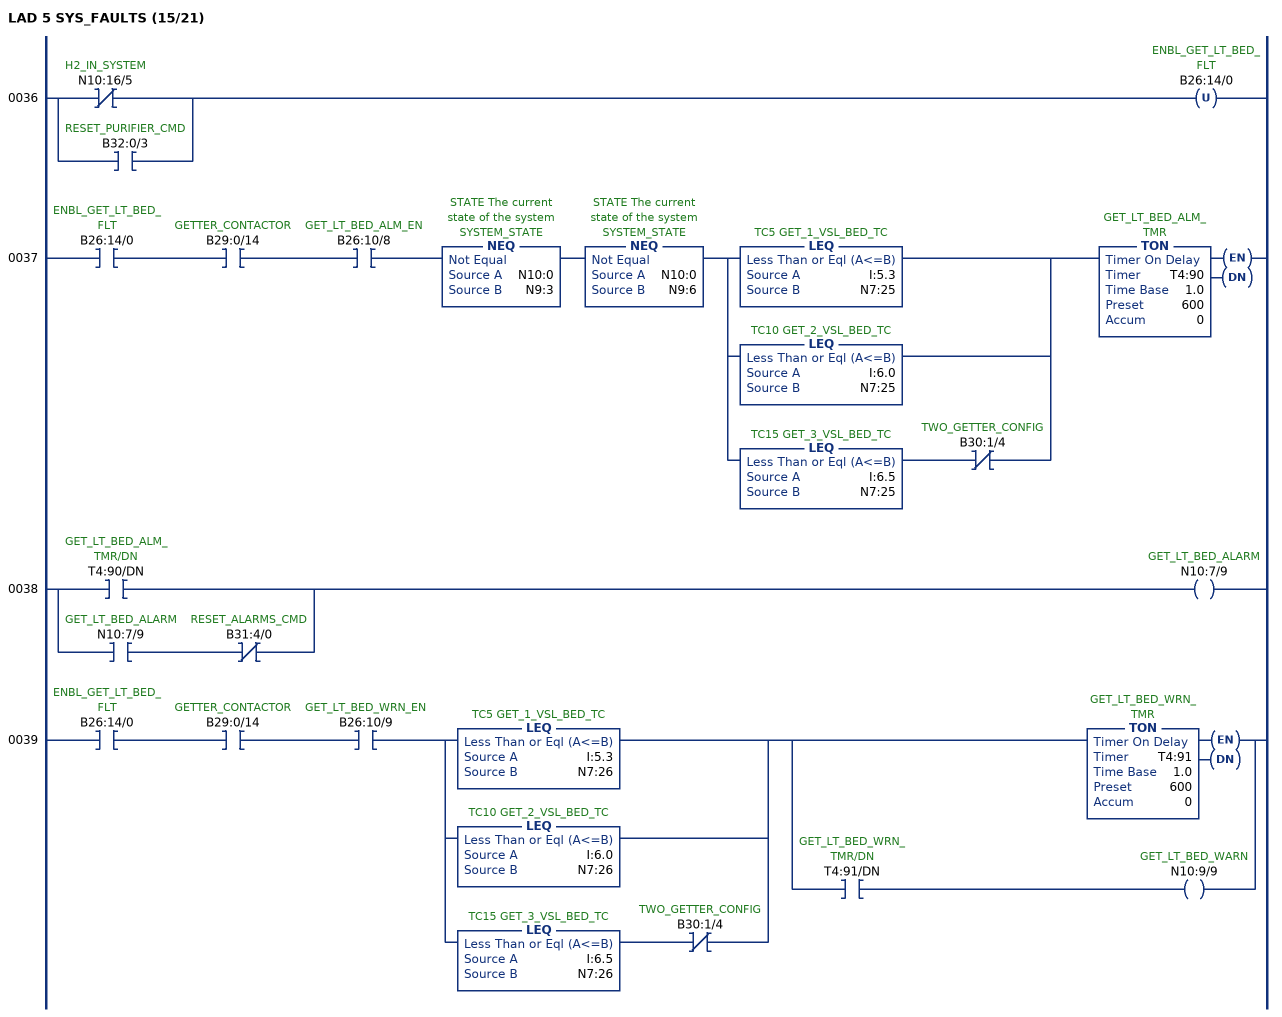
% Rung: 36 %
SOR BST XIO N10:16/5 NXB XIC B32:0/3 BND OTU B26:14/0 EOR
%   N10:16/5  H2_IN_SYSTEM %
%   B32:0/3  RESET_PURIFIER_CMD %
%   B26:14/0  ENBL_GET_LT_BED_FLT %
% Rung: 37 %
SOR XIC B26:14/0 XIC B29:0/14 XIC B26:10/8 NEQ N10:0 N9:3 NEQ N10:0 N9:6 BST LEQ I:5.3 N7:25 NXB LEQ I:6.0 N7:25 NXB LEQ I:6.5 N7:25 XIO B30:1/4 BND TON T4:90 1.0 600 0 EOR
%   B26:14/0  ENBL_GET_LT_BED_FLT %
%   B29:0/14  GETTER_CONTACTOR %
%   B26:10/8  GET_LT_BED_ALM_EN %
%   N10:0  SYSTEM_STATE  "STATE The current state of the system" %
%   N9:3  SYSTEM_MANUAL  "STATE System Manual" %
%   N9:6  SYSTEM_PURGE %
%   I:5.3  GET_1_VSL_BED_TC  "TC5" %
%   N7:25  GET_LT_BED_ALM_SP %
%   I:6.0  GET_2_VSL_BED_TC  "TC10" %
%   I:6.5  GET_3_VSL_BED_TC  "TC15" %
%   B30:1/4  TWO_GETTER_CONFIG %
%   T4:90  GET_LT_BED_ALM_TMR %
% Rung: 38 %
SOR BST XIC T4:90/DN NXB XIC N10:7/9 XIO B31:4/0 BND OTE N10:7/9 EOR
%   T4:90  GET_LT_BED_ALM_TMR %
%   N10:7/9  GET_LT_BED_ALARM %
%   B31:4/0  RESET_ALARMS_CMD %
% Rung: 39 %
SOR XIC B26:14/0 XIC B29:0/14 XIC B26:10/9 BST LEQ I:5.3 N7:26 NXB LEQ I:6.0 N7:26 NXB LEQ I:6.5 N7:26 XIO B30:1/4 BND BST TON T4:91 1.0 600 0 NXB XIC T4:91/DN OTE N10:9/9 BND EOR
%   B26:14/0  ENBL_GET_LT_BED_FLT %
%   B29:0/14  GETTER_CONTACTOR %
%   B26:10/9  GET_LT_BED_WRN_EN %
%   I:5.3  GET_1_VSL_BED_TC  "TC5" %
%   N7:26  GET_LT_BED_WRN_SP %
%   I:6.0  GET_2_VSL_BED_TC  "TC10" %
%   I:6.5  GET_3_VSL_BED_TC  "TC15" %
%   B30:1/4  TWO_GETTER_CONFIG %
%   T4:91  GET_LT_BED_WRN_TMR %
%   N10:9/9  GET_LT_BED_WARN %

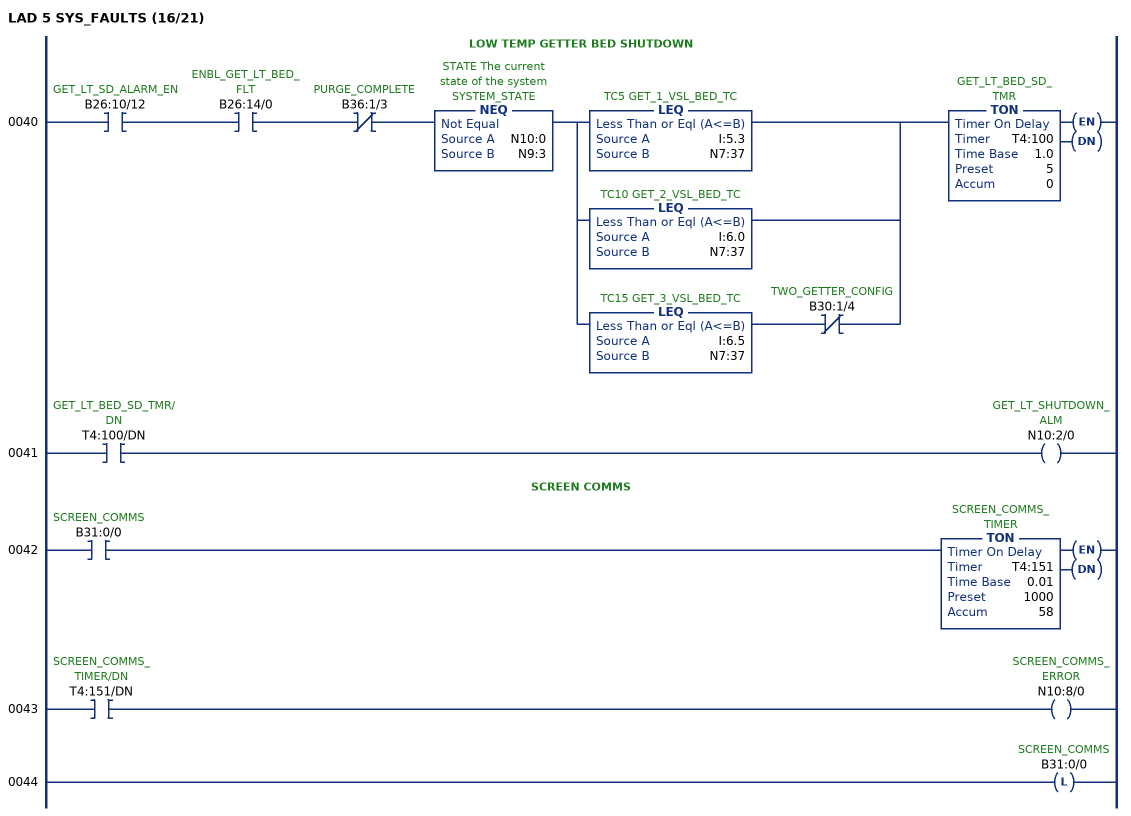
% Rung: 40 %
% TITLE: LOW TEMP GETTER BED SHUTDOWN %
SOR XIC B26:10/12 XIC B26:14/0 XIO B36:1/3 NEQ N10:0 N9:3 BST LEQ I:5.3 N7:37 NXB LEQ I:6.0 N7:37 NXB LEQ I:6.5 N7:37 XIO B30:1/4 BND TON T4:100 1.0 5 0 EOR
%   B26:10/12  GET_LT_SD_ALARM_EN %
%   B26:14/0  ENBL_GET_LT_BED_FLT %
%   B36:1/3  PURGE_COMPLETE %
%   N10:0  SYSTEM_STATE  "STATE The current state of the system" %
%   N9:3  SYSTEM_MANUAL  "STATE System Manual" %
%   I:5.3  GET_1_VSL_BED_TC  "TC5" %
%   N7:37  GET_LT_SHUTDOWN_SP %
%   I:6.0  GET_2_VSL_BED_TC  "TC10" %
%   I:6.5  GET_3_VSL_BED_TC  "TC15" %
%   B30:1/4  TWO_GETTER_CONFIG %
%   T4:100  GET_LT_BED_SD_TMR %
% Rung: 41 %
SOR XIC T4:100/DN OTE N10:2/0 EOR
%   T4:100  GET_LT_BED_SD_TMR %
%   N10:2/0  GET_LT_SHUTDOWN_ALM %
% Rung: 42 %
% TITLE: SCREEN COMMS %
SOR XIC B31:0/0 TON T4:151 0.01 1000 58 EOR
%   B31:0/0  SCREEN_COMMS %
%   T4:151  SCREEN_COMMS_TIMER %
% Rung: 43 %
SOR XIC T4:151/DN OTE N10:8/0 EOR
%   T4:151  SCREEN_COMMS_TIMER %
%   N10:8/0  SCREEN_COMMS_ERROR %
% Rung: 44 %
SOR OTL B31:0/0 EOR
%   B31:0/0  SCREEN_COMMS %

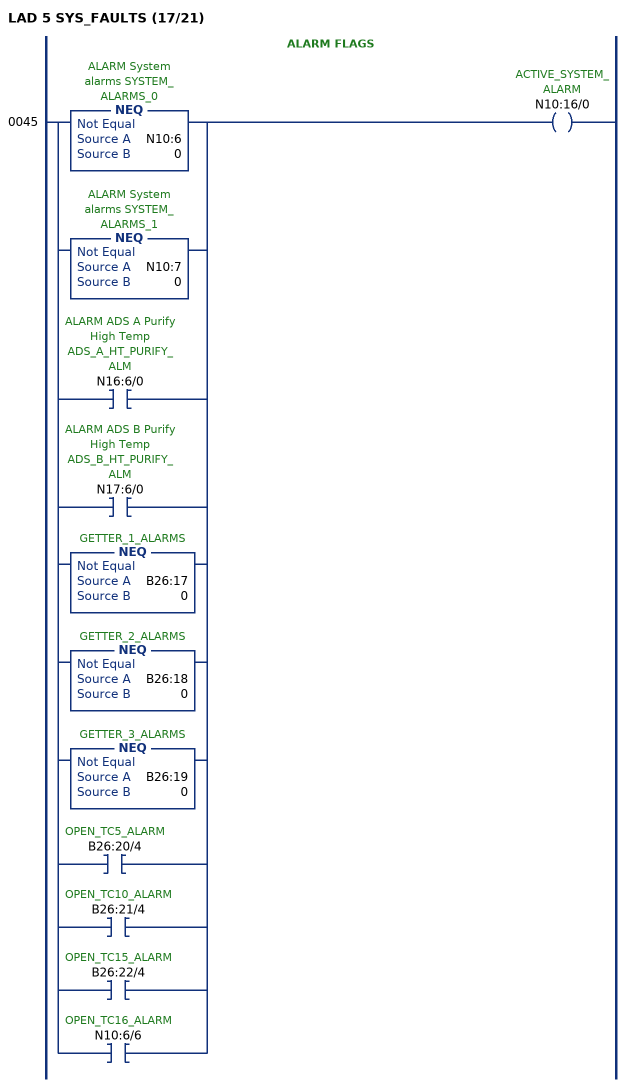
% Rung: 45 %
% TITLE: ALARM FLAGS %
SOR BST NEQ N10:6 0 NXB NEQ N10:7 0 NXB XIC N16:6/0 NXB XIC N17:6/0 NXB NEQ B26:17 0 NXB NEQ B26:18 0 NXB NEQ B26:19 0 NXB XIC B26:20/4 NXB XIC B26:21/4 NXB XIC B26:22/4 NXB XIC N10:6/6 BND OTE N10:16/0 EOR
%   N10:6  SYSTEM_ALARMS_0  "ALARM System alarms" %
%   N10:7  SYSTEM_ALARMS_1  "ALARM System alarms" %
%   N16:6/0  ADS_A_HT_PURIFY_ALM  "ALARM ADS A Purify High Temp" %
%   N17:6/0  ADS_B_HT_PURIFY_ALM  "ALARM ADS B Purify High Temp" %
%   B26:17  GETTER_1_ALARMS %
%   B26:18  GETTER_2_ALARMS %
%   B26:19  GETTER_3_ALARMS %
%   B26:20/4  OPEN_TC5_ALARM %
%   B26:21/4  OPEN_TC10_ALARM %
%   B26:22/4  OPEN_TC15_ALARM %
%   N10:6/6  OPEN_TC16_ALARM %
%   N10:16/0  ACTIVE_SYSTEM_ALARM %

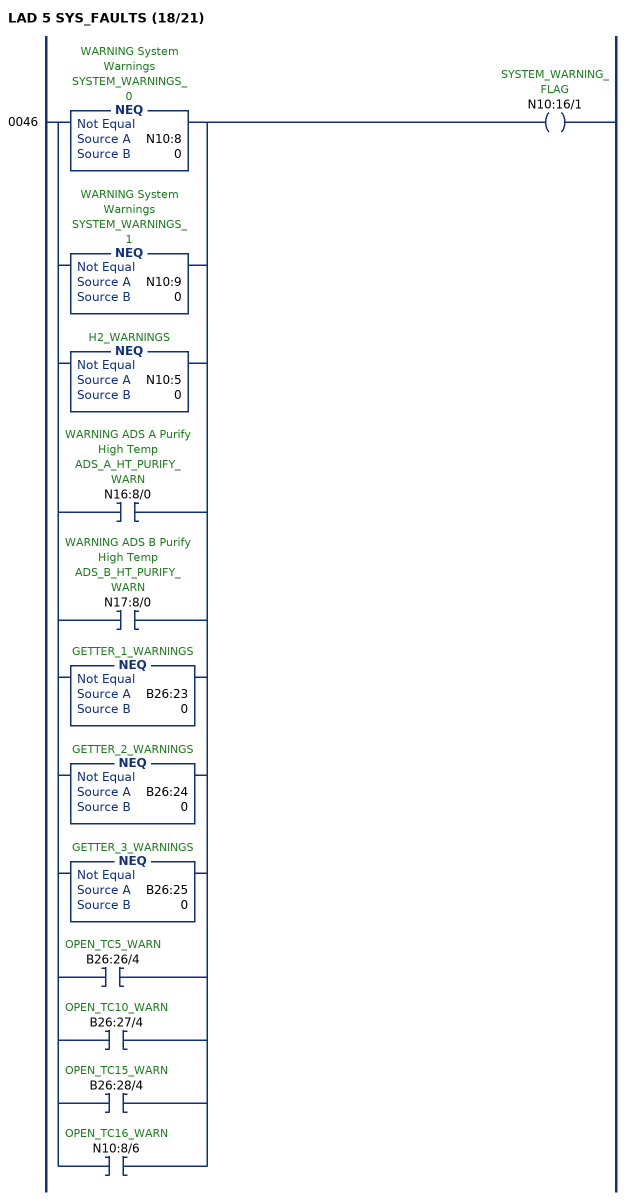
% Rung: 46 %
SOR BST NEQ N10:8 0 NXB NEQ N10:9 0 NXB NEQ N10:5 0 NXB XIC N16:8/0 NXB XIC N17:8/0 NXB NEQ B26:23 0 NXB NEQ B26:24 0 NXB NEQ B26:25 0 NXB XIC B26:26/4 NXB XIC B26:27/4 NXB XIC B26:28/4 NXB XIC N10:8/6 BND OTE N10:16/1 EOR
%   N10:8  SYSTEM_WARNINGS_0  "WARNING System Warnings" %
%   N10:9  SYSTEM_WARNINGS_1  "WARNING System Warnings" %
%   N10:5  H2_WARNINGS %
%   N16:8/0  ADS_A_HT_PURIFY_WARN  "WARNING ADS A Purify High Temp" %
%   N17:8/0  ADS_B_HT_PURIFY_WARN  "WARNING ADS B Purify High Temp" %
%   B26:23  GETTER_1_WARNINGS %
%   B26:24  GETTER_2_WARNINGS %
%   B26:25  GETTER_3_WARNINGS %
%   B26:26/4  OPEN_TC5_WARN %
%   B26:27/4  OPEN_TC10_WARN %
%   B26:28/4  OPEN_TC15_WARN %
%   N10:8/6  OPEN_TC16_WARN %
%   N10:16/1  SYSTEM_WARNING_FLAG %

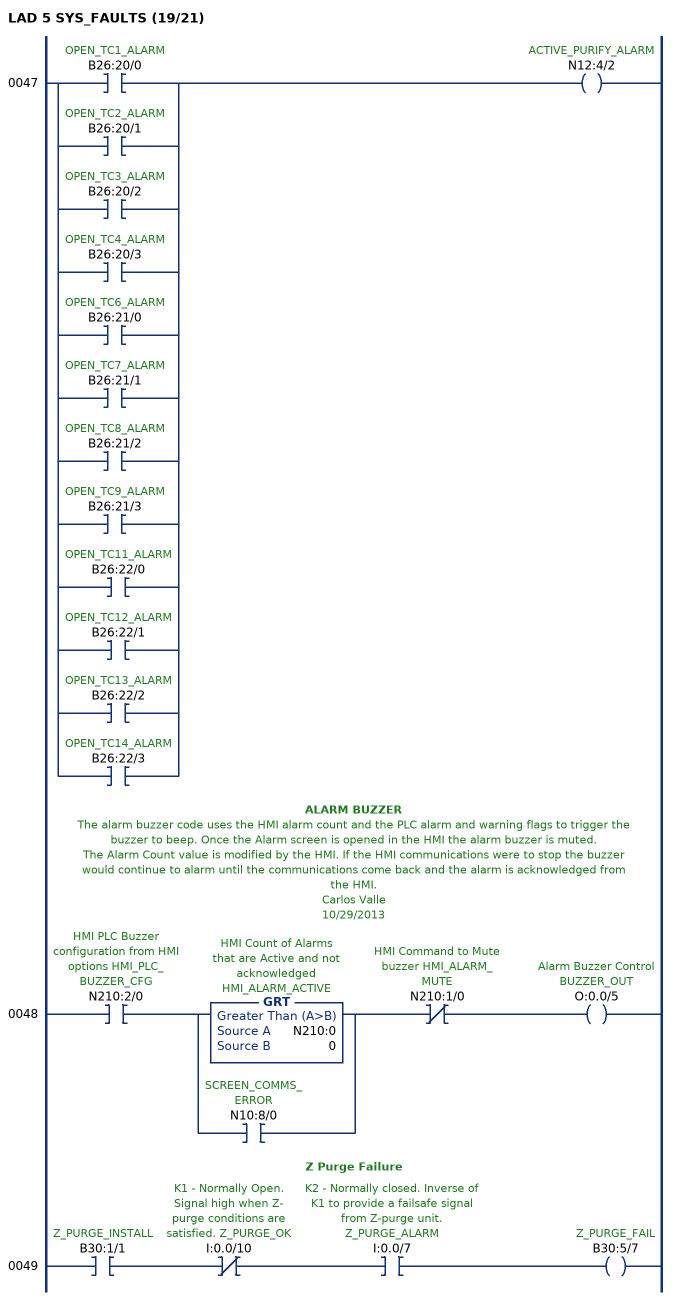
% Rung: 47 %
SOR BST XIC B26:20/0 NXB XIC B26:20/1 NXB XIC B26:20/2 NXB XIC B26:20/3 NXB XIC B26:21/0 NXB XIC B26:21/1 NXB XIC B26:21/2 NXB XIC B26:21/3 NXB XIC B26:22/0 NXB XIC B26:22/1 NXB XIC B26:22/2 NXB XIC B26:22/3 BND OTE N12:4/2 EOR
%   B26:20/0  OPEN_TC1_ALARM %
%   B26:20/1  OPEN_TC2_ALARM %
%   B26:20/2  OPEN_TC3_ALARM %
%   B26:20/3  OPEN_TC4_ALARM %
%   B26:21/0  OPEN_TC6_ALARM %
%   B26:21/1  OPEN_TC7_ALARM %
%   B26:21/2  OPEN_TC8_ALARM %
%   B26:21/3  OPEN_TC9_ALARM %
%   B26:22/0  OPEN_TC11_ALARM %
%   B26:22/1  OPEN_TC12_ALARM %
%   B26:22/2  OPEN_TC13_ALARM %
%   B26:22/3  OPEN_TC14_ALARM %
%   N12:4/2  ACTIVE_PURIFY_ALARM %
% Rung: 48 %
% TITLE: ALARM BUZZER %
% The alarm buzzer code uses the HMI alarm count and the PLC alarm and warning flags to trigger the buzzer to beep. Once the Alarm screen is opened in the HMI the alarm buzzer is muted.
% The Alarm Count value is modified by the HMI. If the HMI communications were to stop the buzzer would continue to alarm until the communications come back and the alarm is acknowledged from the HMI.
% Carlos Valle
% 10/29/2013 %
SOR XIC N210:2/0 BST GRT N210:0 0 NXB XIC N10:8/0 BND XIO N210:1/0 OTE O:0.0/5 EOR
%   N210:2/0  HMI_PLC_BUZZER_CFG  "HMI PLC Buzzer configuration from HMI options" %
%   N210:0  HMI_ALARM_ACTIVE  "HMI Count of Alarms that are Active and not acknowledged" %
%   N10:8/0  SCREEN_COMMS_ERROR %
%   N210:1/0  HMI_ALARM_MUTE  "HMI Command to Mute buzzer" %
%   O:0.0/5  BUZZER_OUT  "Alarm Buzzer Control" %
% Rung: 49 %
% TITLE: Z Purge Failure %
SOR XIC B30:1/1 XIO I:0.0/10 XIC I:0.0/7 OTE B30:5/7 EOR
%   B30:1/1  Z_PURGE_INSTALL %
%   I:0.0/10  Z_PURGE_OK  "K1 - Normally Open. Signal high when Z- purge conditions are satisfied." %
%   I:0.0/7  Z_PURGE_ALARM  "K2 - Normally closed. Inverse of K1 to provide a failsafe signal from Z-purge unit." %
%   B30:5/7  Z_PURGE_FAIL %

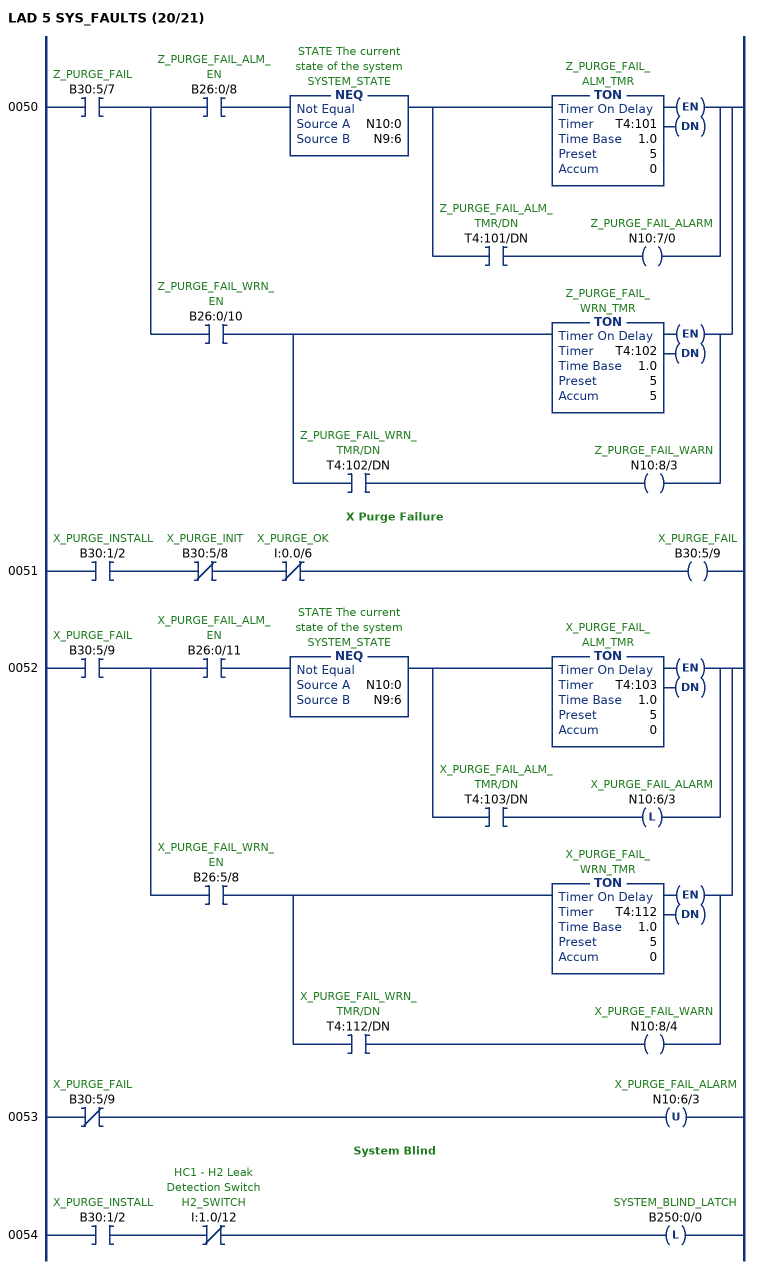
% Rung: 50 %
SOR XIC B30:5/7 BST XIC B26:0/8 NEQ N10:0 N9:6 BST TON T4:101 1.0 5 0 NXB XIC T4:101/DN OTE N10:7/0 BND NXB XIC B26:0/10 BST TON T4:102 1.0 5 5 NXB XIC T4:102/DN OTE N10:8/3 BND BND EOR
%   B30:5/7  Z_PURGE_FAIL %
%   B26:0/8  Z_PURGE_FAIL_ALM_EN %
%   N10:0  SYSTEM_STATE  "STATE The current state of the system" %
%   N9:6  SYSTEM_PURGE %
%   T4:101  Z_PURGE_FAIL_ALM_TMR %
%   N10:7/0  Z_PURGE_FAIL_ALARM %
%   B26:0/10  Z_PURGE_FAIL_WRN_EN %
%   T4:102  Z_PURGE_FAIL_WRN_TMR %
%   N10:8/3  Z_PURGE_FAIL_WARN %
% Rung: 51 %
% TITLE: X Purge Failure %
SOR XIC B30:1/2 XIO B30:5/8 XIO I:0.0/6 OTE B30:5/9 EOR
%   B30:1/2  X_PURGE_INSTALL %
%   B30:5/8  X_PURGE_INIT %
%   I:0.0/6  X_PURGE_OK %
%   B30:5/9  X_PURGE_FAIL %
% Rung: 52 %
SOR XIC B30:5/9 BST XIC B26:0/11 NEQ N10:0 N9:6 BST TON T4:103 1.0 5 0 NXB XIC T4:103/DN OTL N10:6/3 BND NXB XIC B26:5/8 BST TON T4:112 1.0 5 0 NXB XIC T4:112/DN OTE N10:8/4 BND BND EOR
%   B30:5/9  X_PURGE_FAIL %
%   B26:0/11  X_PURGE_FAIL_ALM_EN %
%   N10:0  SYSTEM_STATE  "STATE The current state of the system" %
%   N9:6  SYSTEM_PURGE %
%   T4:103  X_PURGE_FAIL_ALM_TMR %
%   N10:6/3  X_PURGE_FAIL_ALARM %
%   B26:5/8  X_PURGE_FAIL_WRN_EN %
%   T4:112  X_PURGE_FAIL_WRN_TMR %
%   N10:8/4  X_PURGE_FAIL_WARN %
% Rung: 53 %
SOR XIO B30:5/9 OTU N10:6/3 EOR
%   B30:5/9  X_PURGE_FAIL %
%   N10:6/3  X_PURGE_FAIL_ALARM %
% Rung: 54 %
% TITLE: System Blind %
SOR XIC B30:1/2 XIO I:1.0/12 OTL B250:0/0 EOR
%   B30:1/2  X_PURGE_INSTALL %
%   I:1.0/12  H2_SWITCH  "HC1 - H2 Leak Detection Switch" %
%   B250:0/0  SYSTEM_BLIND_LATCH %

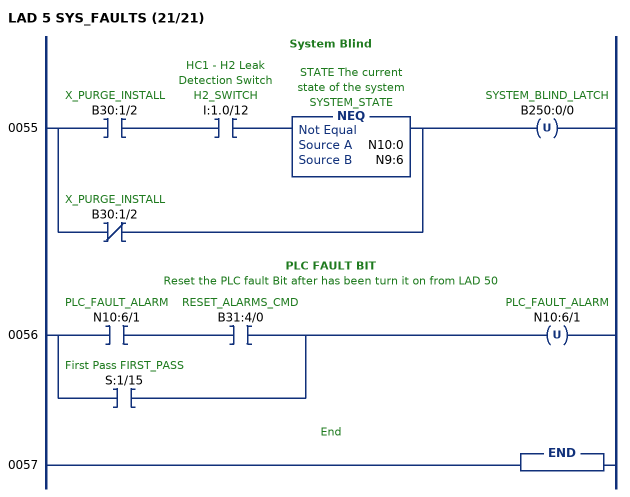
% Rung: 55 %
% TITLE: System Blind %
SOR BST XIC B30:1/2 XIC I:1.0/12 NEQ N10:0 N9:6 NXB XIO B30:1/2 BND OTU B250:0/0 EOR
%   B30:1/2  X_PURGE_INSTALL %
%   I:1.0/12  H2_SWITCH  "HC1 - H2 Leak Detection Switch" %
%   N10:0  SYSTEM_STATE  "STATE The current state of the system" %
%   N9:6  SYSTEM_PURGE %
%   B250:0/0  SYSTEM_BLIND_LATCH %
% Rung: 56 %
% TITLE: PLC FAULT BIT %
% Reset the PLC fault Bit after has been turn it on from LAD 50 %
SOR BST XIC N10:6/1 XIC B31:4/0 NXB XIC S:1/15 BND OTU N10:6/1 EOR
%   N10:6/1  PLC_FAULT_ALARM %
%   B31:4/0  RESET_ALARMS_CMD %
%   S:1/15  FIRST_PASS  "First Pass" %
% Rung: 57 %
% End %
SOR END EOR

LADDER 6 "SYSTEM"    % Controls the system %
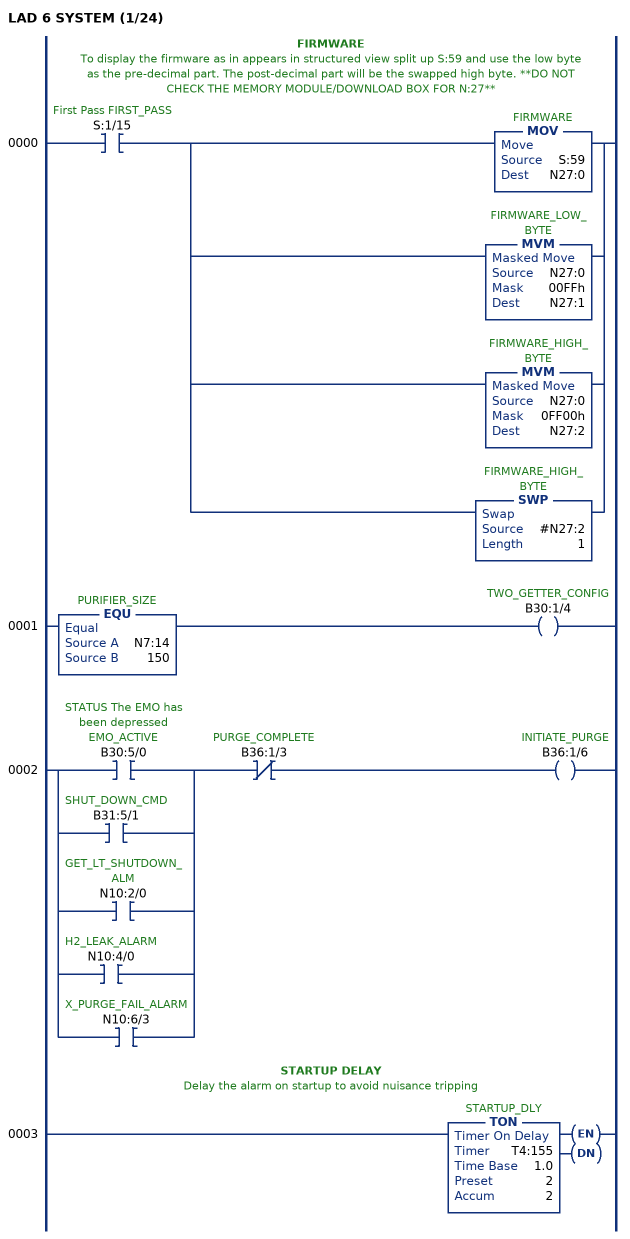
% Rung: 0 %
% TITLE: FIRMWARE %
% To display the firmware as in appears in structured view split up S:59 and use the low byte as the pre-decimal part. The post-decimal part will be the swapped high byte. **DO NOT CHECK THE MEMORY MODULE/DOWNLOAD BOX FOR N:27** %
SOR XIC S:1/15 BST MOV S:59 N27:0 NXB MVM N27:0 00FFh N27:1 NXB MVM N27:0 0FF00h N27:2 NXB SWP #N27:2 1 BND EOR
%   S:1/15  FIRST_PASS  "First Pass" %
%   S:59  "Operating System FRN" %
%   N27:0  FIRMWARE %
%   N27:1  FIRMWARE_LOW_BYTE %
%   N27:2  FIRMWARE_HIGH_BYTE %
% Rung: 1 %
SOR EQU N7:14 150 OTE B30:1/4 EOR
%   N7:14  PURIFIER_SIZE %
%   B30:1/4  TWO_GETTER_CONFIG %
% Rung: 2 %
SOR BST XIC B30:5/0 NXB XIC B31:5/1 NXB XIC N10:2/0 NXB XIC N10:4/0 NXB XIC N10:6/3 BND XIO B36:1/3 OTE B36:1/6 EOR
%   B30:5/0  EMO_ACTIVE  "STATUS The EMO has been depressed" %
%   B31:5/1  SHUT_DOWN_CMD %
%   N10:2/0  GET_LT_SHUTDOWN_ALM %
%   N10:4/0  H2_LEAK_ALARM %
%   N10:6/3  X_PURGE_FAIL_ALARM %
%   B36:1/3  PURGE_COMPLETE %
%   B36:1/6  INITIATE_PURGE %
% Rung: 3 %
% TITLE: STARTUP DELAY %
% Delay the alarm on startup to avoid nuisance tripping %
SOR TON T4:155 1.0 2 2 EOR
%   T4:155  STARTUP_DLY %

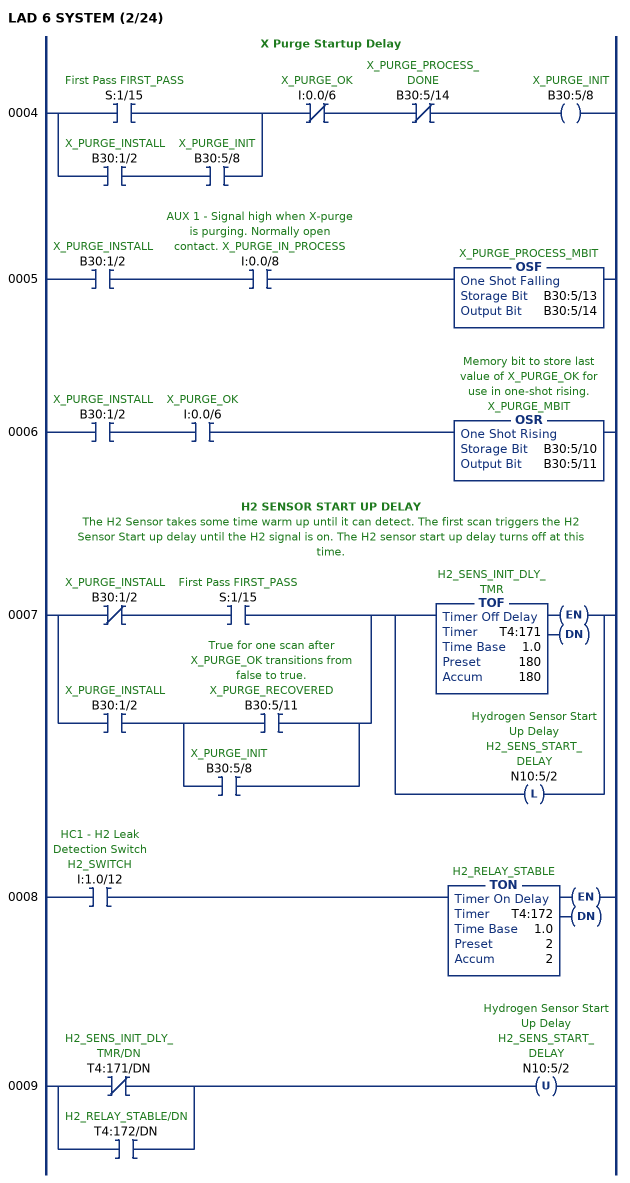
% Rung: 4 %
% TITLE: X Purge Startup Delay %
SOR BST XIC S:1/15 NXB XIC B30:1/2 XIC B30:5/8 BND XIO I:0.0/6 XIO B30:5/14 OTE B30:5/8 EOR
%   S:1/15  FIRST_PASS  "First Pass" %
%   B30:1/2  X_PURGE_INSTALL %
%   B30:5/8  X_PURGE_INIT %
%   I:0.0/6  X_PURGE_OK %
%   B30:5/14  X_PURGE_PROCESS_DONE %
% Rung: 5 %
SOR XIC B30:1/2 XIC I:0.0/8 OSF B30:5/13 B30:5/14 EOR
%   B30:1/2  X_PURGE_INSTALL %
%   I:0.0/8  X_PURGE_IN_PROCESS  "AUX 1 - Signal high when X-purge is purging. Normally open contact." %
%   B30:5/13  X_PURGE_PROCESS_MBIT %
%   B30:5/14  X_PURGE_PROCESS_DONE %
% Rung: 6 %
SOR XIC B30:1/2 XIC I:0.0/6 OSR B30:5/10 B30:5/11 EOR
%   B30:1/2  X_PURGE_INSTALL %
%   I:0.0/6  X_PURGE_OK %
%   B30:5/10  X_PURGE_MBIT  "Memory bit to store last value of X_PURGE_OK for use in one-shot rising." %
%   B30:5/11  X_PURGE_RECOVERED  "True for one scan after X_PURGE_OK transitions from false to true." %
% Rung: 7 %
% TITLE: H2 SENSOR START UP DELAY %
% The H2 Sensor takes some time warm up until it can detect. The first scan triggers the H2 Sensor Start up delay until the H2 signal is on. The H2 sensor start up delay turns off at this time. %
SOR BST XIO B30:1/2 XIC S:1/15 NXB XIC B30:1/2 BST XIC B30:5/11 NXB XIC B30:5/8 BND BND BST TOF T4:171 1.0 180 180 NXB OTL N10:5/2 BND EOR
%   B30:1/2  X_PURGE_INSTALL %
%   S:1/15  FIRST_PASS  "First Pass" %
%   B30:5/11  X_PURGE_RECOVERED  "True for one scan after X_PURGE_OK transitions from false to true." %
%   B30:5/8  X_PURGE_INIT %
%   T4:171  H2_SENS_INIT_DLY_TMR %
%   N10:5/2  H2_SENS_START_DELAY  "Hydrogen Sensor Start Up Delay" %
% Rung: 8 %
SOR XIC I:1.0/12 TON T4:172 1.0 2 2 EOR
%   I:1.0/12  H2_SWITCH  "HC1 - H2 Leak Detection Switch" %
%   T4:172  H2_RELAY_STABLE %
% Rung: 9 %
SOR BST XIO T4:171/DN NXB XIC T4:172/DN BND OTU N10:5/2 EOR
%   T4:171  H2_SENS_INIT_DLY_TMR %
%   T4:172  H2_RELAY_STABLE %
%   N10:5/2  H2_SENS_START_DELAY  "Hydrogen Sensor Start Up Delay" %

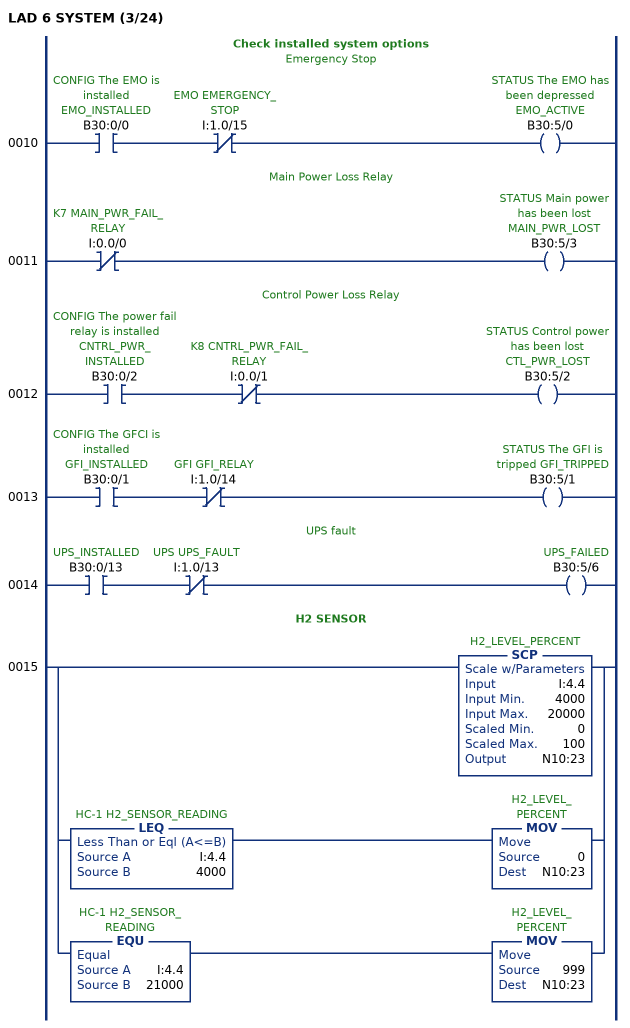
% Rung: 10 %
% TITLE: Check installed system options %
% Emergency Stop %
SOR XIC B30:0/0 XIO I:1.0/15 OTE B30:5/0 EOR
%   B30:0/0  EMO_INSTALLED  "CONFIG The EMO is installed" %
%   I:1.0/15  EMERGENCY_STOP  "EMO" %
%   B30:5/0  EMO_ACTIVE  "STATUS The EMO has been depressed" %
% Rung: 11 %
% Main Power Loss Relay %
SOR XIO I:0.0/0 OTE B30:5/3 EOR
%   I:0.0/0  MAIN_PWR_FAIL_RELAY  "K7" %
%   B30:5/3  MAIN_PWR_LOST  "STATUS Main power has been lost" %
% Rung: 12 %
% Control Power Loss Relay %
SOR XIC B30:0/2 XIO I:0.0/1 OTE B30:5/2 EOR
%   B30:0/2  CNTRL_PWR_INSTALLED  "CONFIG The power fail relay is installed" %
%   I:0.0/1  CNTRL_PWR_FAIL_RELAY  "K8" %
%   B30:5/2  CTL_PWR_LOST  "STATUS Control power has been lost" %
% Rung: 13 %
SOR XIC B30:0/1 XIO I:1.0/14 OTE B30:5/1 EOR
%   B30:0/1  GFI_INSTALLED  "CONFIG The GFCI is installed" %
%   I:1.0/14  GFI_RELAY  "GFI" %
%   B30:5/1  GFI_TRIPPED  "STATUS The GFI is tripped" %
% Rung: 14 %
% UPS fault %
SOR XIC B30:0/13 XIO I:1.0/13 OTE B30:5/6 EOR
%   B30:0/13  UPS_INSTALLED %
%   I:1.0/13  UPS_FAULT  "UPS" %
%   B30:5/6  UPS_FAILED %
% Rung: 15 %
% TITLE: H2 SENSOR %
SOR BST SCP I:4.4 4000 20000 0 100 N10:23 NXB LEQ I:4.4 4000 MOV 0 N10:23 NXB EQU I:4.4 21000 MOV 999 N10:23 BND EOR
%   I:4.4  H2_SENSOR_READING  "HC-1" %
%   N10:23  H2_LEVEL_PERCENT %

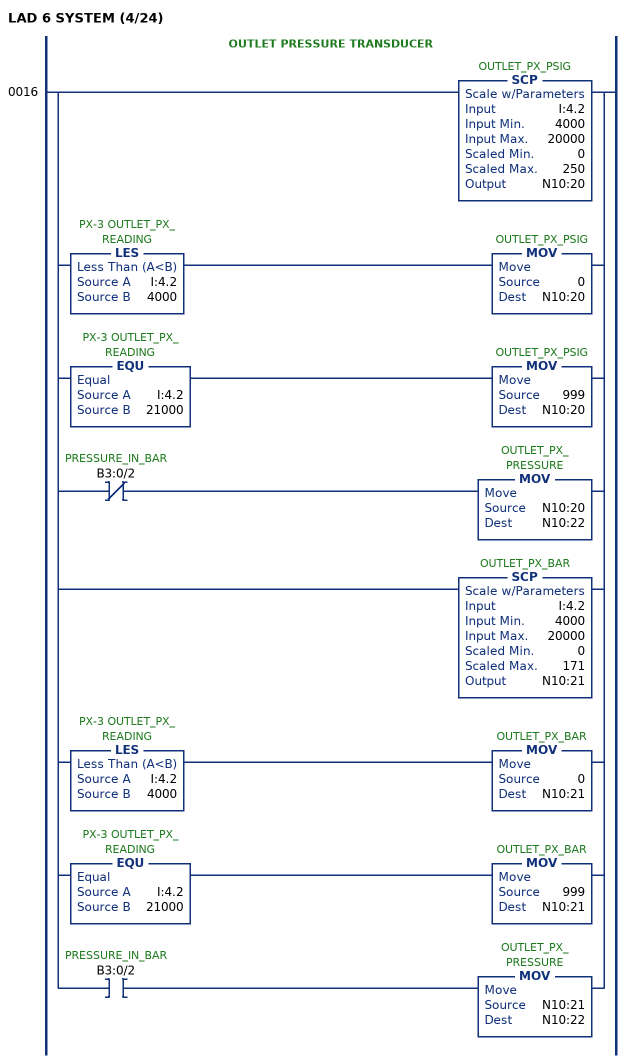
% Rung: 16 %
% TITLE: OUTLET PRESSURE TRANSDUCER %
SOR BST SCP I:4.2 4000 20000 0 250 N10:20 NXB LES I:4.2 4000 MOV 0 N10:20 NXB EQU I:4.2 21000 MOV 999 N10:20 NXB XIO B3:0/2 MOV N10:20 N10:22 NXB SCP I:4.2 4000 20000 0 171 N10:21 NXB LES I:4.2 4000 MOV 0 N10:21 NXB EQU I:4.2 21000 MOV 999 N10:21 NXB XIC B3:0/2 MOV N10:21 N10:22 BND EOR
%   I:4.2  OUTLET_PX_READING  "PX-3" %
%   N10:20  OUTLET_PX_PSIG %
%   B3:0/2  PRESSURE_IN_BAR %
%   N10:22  OUTLET_PX_PRESSURE %
%   N10:21  OUTLET_PX_BAR %

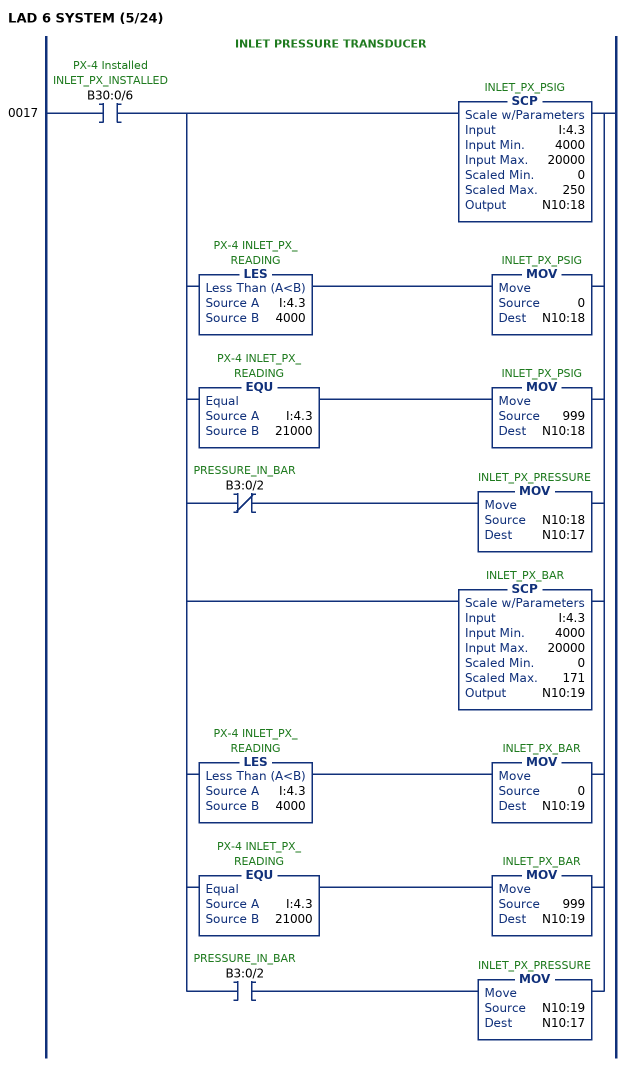
% Rung: 17 %
% TITLE: INLET PRESSURE TRANSDUCER %
SOR XIC B30:0/6 BST SCP I:4.3 4000 20000 0 250 N10:18 NXB LES I:4.3 4000 MOV 0 N10:18 NXB EQU I:4.3 21000 MOV 999 N10:18 NXB XIO B3:0/2 MOV N10:18 N10:17 NXB SCP I:4.3 4000 20000 0 171 N10:19 NXB LES I:4.3 4000 MOV 0 N10:19 NXB EQU I:4.3 21000 MOV 999 N10:19 NXB XIC B3:0/2 MOV N10:19 N10:17 BND EOR
%   B30:0/6  INLET_PX_INSTALLED  "PX-4 Installed" %
%   I:4.3  INLET_PX_READING  "PX-4" %
%   N10:18  INLET_PX_PSIG %
%   B3:0/2  PRESSURE_IN_BAR %
%   N10:17  INLET_PX_PRESSURE %
%   N10:19  INLET_PX_BAR %

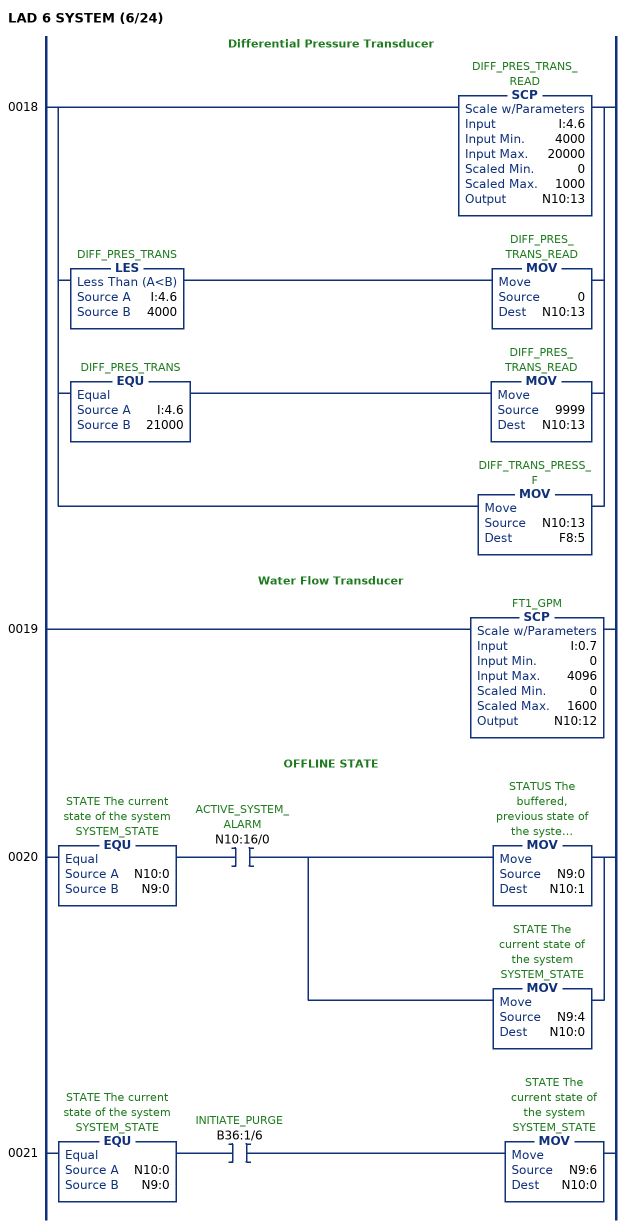
% Rung: 18 %
% TITLE: Differential Pressure Transducer %
SOR BST SCP I:4.6 4000 20000 0 1000 N10:13 NXB LES I:4.6 4000 MOV 0 N10:13 NXB EQU I:4.6 21000 MOV 9999 N10:13 NXB MOV N10:13 F8:5 BND EOR
%   I:4.6  DIFF_PRES_TRANS %
%   N10:13  DIFF_PRES_TRANS_READ %
%   F8:5  DIFF_TRANS_PRESS_F %
% Rung: 19 %
% TITLE: Water Flow Transducer %
SOR SCP I:0.7 0 4096 0 1600 N10:12 EOR
%   I:0.7  WATER_FLOW_TDX_FT1 %
%   N10:12  FT1_GPM %
% Rung: 20 %
% TITLE: OFFLINE STATE %
SOR EQU N10:0 N9:0 XIC N10:16/0 BST MOV N9:0 N10:1 NXB MOV N9:4 N10:0 BND EOR
%   N10:0  SYSTEM_STATE  "STATE The current state of the system" %
%   N9:0  SYSTEM_OFFLINE %
%   N10:16/0  ACTIVE_SYSTEM_ALARM %
%   N10:1  SYSTEM_STATE_BUFFER  "STATUS The buffered, previous state of the system" %
%   N9:4  SYSTEM_ALARM  "STATE System Alarm" %
% Rung: 21 %
SOR EQU N10:0 N9:0 XIC B36:1/6 MOV N9:6 N10:0 EOR
%   N10:0  SYSTEM_STATE  "STATE The current state of the system" %
%   N9:0  SYSTEM_OFFLINE %
%   B36:1/6  INITIATE_PURGE %
%   N9:6  SYSTEM_PURGE %

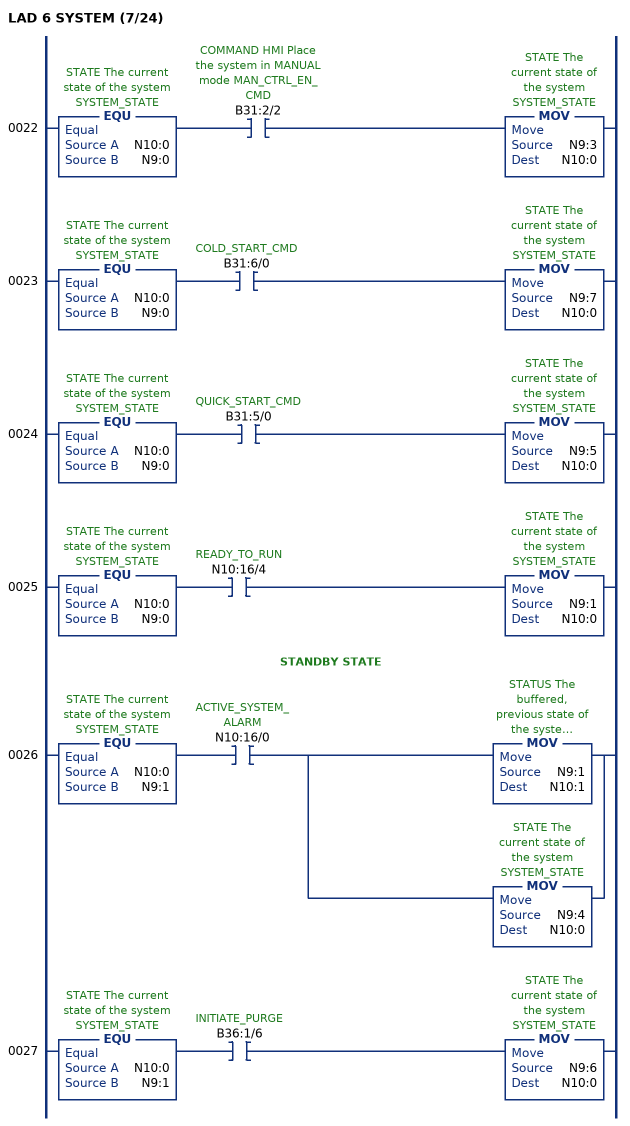
% Rung: 22 %
SOR EQU N10:0 N9:0 XIC B31:2/2 MOV N9:3 N10:0 EOR
%   N10:0  SYSTEM_STATE  "STATE The current state of the system" %
%   N9:0  SYSTEM_OFFLINE %
%   B31:2/2  MAN_CTRL_EN_CMD  "COMMAND HMI Place the system in MANUAL mode" %
%   N9:3  SYSTEM_MANUAL  "STATE System Manual" %
% Rung: 23 %
SOR EQU N10:0 N9:0 XIC B31:6/0 MOV N9:7 N10:0 EOR
%   N10:0  SYSTEM_STATE  "STATE The current state of the system" %
%   N9:0  SYSTEM_OFFLINE %
%   B31:6/0  COLD_START_CMD %
%   N9:7  SYSTEM_COLD_START %
% Rung: 24 %
SOR EQU N10:0 N9:0 XIC B31:5/0 MOV N9:5 N10:0 EOR
%   N10:0  SYSTEM_STATE  "STATE The current state of the system" %
%   N9:0  SYSTEM_OFFLINE %
%   B31:5/0  QUICK_START_CMD %
%   N9:5  SYSTEM_QUICK_START %
% Rung: 25 %
SOR EQU N10:0 N9:0 XIC N10:16/4 MOV N9:1 N10:0 EOR
%   N10:0  SYSTEM_STATE  "STATE The current state of the system" %
%   N9:0  SYSTEM_OFFLINE %
%   N10:16/4  READY_TO_RUN %
%   N9:1  SYSTEM_STANDBY  "STATE System Process" %
% Rung: 26 %
% TITLE: STANDBY STATE %
SOR EQU N10:0 N9:1 XIC N10:16/0 BST MOV N9:1 N10:1 NXB MOV N9:4 N10:0 BND EOR
%   N10:0  SYSTEM_STATE  "STATE The current state of the system" %
%   N9:1  SYSTEM_STANDBY  "STATE System Process" %
%   N10:16/0  ACTIVE_SYSTEM_ALARM %
%   N10:1  SYSTEM_STATE_BUFFER  "STATUS The buffered, previous state of the system" %
%   N9:4  SYSTEM_ALARM  "STATE System Alarm" %
% Rung: 27 %
SOR EQU N10:0 N9:1 XIC B36:1/6 MOV N9:6 N10:0 EOR
%   N10:0  SYSTEM_STATE  "STATE The current state of the system" %
%   N9:1  SYSTEM_STANDBY  "STATE System Process" %
%   B36:1/6  INITIATE_PURGE %
%   N9:6  SYSTEM_PURGE %

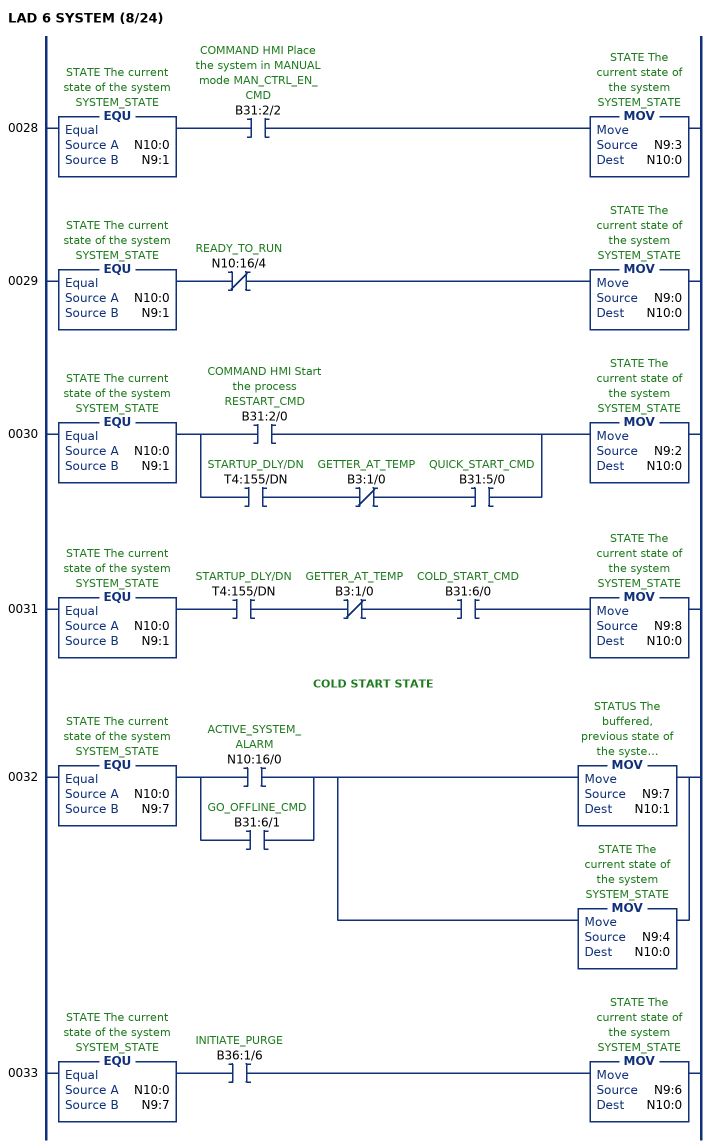
% Rung: 28 %
SOR EQU N10:0 N9:1 XIC B31:2/2 MOV N9:3 N10:0 EOR
%   N10:0  SYSTEM_STATE  "STATE The current state of the system" %
%   N9:1  SYSTEM_STANDBY  "STATE System Process" %
%   B31:2/2  MAN_CTRL_EN_CMD  "COMMAND HMI Place the system in MANUAL mode" %
%   N9:3  SYSTEM_MANUAL  "STATE System Manual" %
% Rung: 29 %
SOR EQU N10:0 N9:1 XIO N10:16/4 MOV N9:0 N10:0 EOR
%   N10:0  SYSTEM_STATE  "STATE The current state of the system" %
%   N9:1  SYSTEM_STANDBY  "STATE System Process" %
%   N10:16/4  READY_TO_RUN %
%   N9:0  SYSTEM_OFFLINE %
% Rung: 30 %
SOR EQU N10:0 N9:1 BST XIC B31:2/0 NXB XIC T4:155/DN XIO B3:1/0 XIC B31:5/0 BND MOV N9:2 N10:0 EOR
%   N10:0  SYSTEM_STATE  "STATE The current state of the system" %
%   N9:1  SYSTEM_STANDBY  "STATE System Process" %
%   B31:2/0  RESTART_CMD  "COMMAND HMI Start the process" %
%   T4:155  STARTUP_DLY %
%   B3:1/0  GETTER_AT_TEMP %
%   B31:5/0  QUICK_START_CMD %
%   N9:2  SYSTEM_PROCESS  "STATE System Process" %
% Rung: 31 %
SOR EQU N10:0 N9:1 XIC T4:155/DN XIO B3:1/0 XIC B31:6/0 MOV N9:8 N10:0 EOR
%   N10:0  SYSTEM_STATE  "STATE The current state of the system" %
%   N9:1  SYSTEM_STANDBY  "STATE System Process" %
%   T4:155  STARTUP_DLY %
%   B3:1/0  GETTER_AT_TEMP %
%   B31:6/0  COLD_START_CMD %
%   N9:8  SYSTEM_SUPPLEMENTAL %
% Rung: 32 %
% TITLE: COLD START STATE %
SOR EQU N10:0 N9:7 BST XIC N10:16/0 NXB XIC B31:6/1 BND BST MOV N9:7 N10:1 NXB MOV N9:4 N10:0 BND EOR
%   N10:0  SYSTEM_STATE  "STATE The current state of the system" %
%   N9:7  SYSTEM_COLD_START %
%   N10:16/0  ACTIVE_SYSTEM_ALARM %
%   B31:6/1  GO_OFFLINE_CMD %
%   N10:1  SYSTEM_STATE_BUFFER  "STATUS The buffered, previous state of the system" %
%   N9:4  SYSTEM_ALARM  "STATE System Alarm" %
% Rung: 33 %
SOR EQU N10:0 N9:7 XIC B36:1/6 MOV N9:6 N10:0 EOR
%   N10:0  SYSTEM_STATE  "STATE The current state of the system" %
%   N9:7  SYSTEM_COLD_START %
%   B36:1/6  INITIATE_PURGE %
%   N9:6  SYSTEM_PURGE %

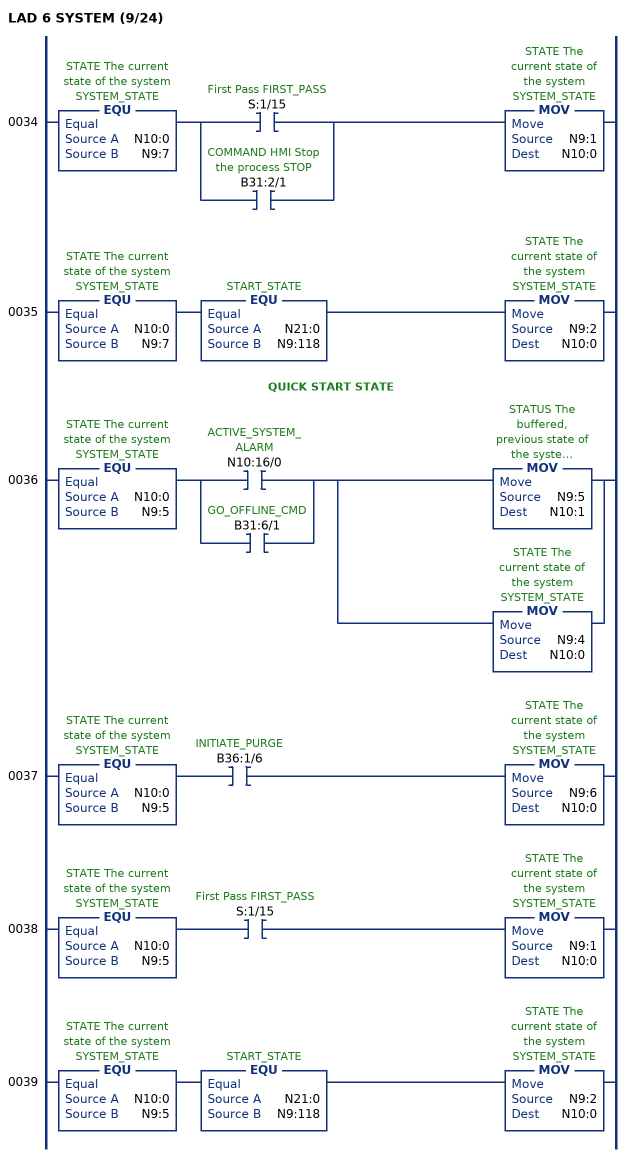
% Rung: 34 %
SOR EQU N10:0 N9:7 BST XIC S:1/15 NXB XIC B31:2/1 BND MOV N9:1 N10:0 EOR
%   N10:0  SYSTEM_STATE  "STATE The current state of the system" %
%   N9:7  SYSTEM_COLD_START %
%   S:1/15  FIRST_PASS  "First Pass" %
%   B31:2/1  STOP  "COMMAND HMI Stop the process" %
%   N9:1  SYSTEM_STANDBY  "STATE System Process" %
% Rung: 35 %
SOR EQU N10:0 N9:7 EQU N21:0 N9:118 MOV N9:2 N10:0 EOR
%   N10:0  SYSTEM_STATE  "STATE The current state of the system" %
%   N9:7  SYSTEM_COLD_START %
%   N21:0  START_STATE %
%   N9:118  START_DONE %
%   N9:2  SYSTEM_PROCESS  "STATE System Process" %
% Rung: 36 %
% TITLE: QUICK START STATE %
SOR EQU N10:0 N9:5 BST XIC N10:16/0 NXB XIC B31:6/1 BND BST MOV N9:5 N10:1 NXB MOV N9:4 N10:0 BND EOR
%   N10:0  SYSTEM_STATE  "STATE The current state of the system" %
%   N9:5  SYSTEM_QUICK_START %
%   N10:16/0  ACTIVE_SYSTEM_ALARM %
%   B31:6/1  GO_OFFLINE_CMD %
%   N10:1  SYSTEM_STATE_BUFFER  "STATUS The buffered, previous state of the system" %
%   N9:4  SYSTEM_ALARM  "STATE System Alarm" %
% Rung: 37 %
SOR EQU N10:0 N9:5 XIC B36:1/6 MOV N9:6 N10:0 EOR
%   N10:0  SYSTEM_STATE  "STATE The current state of the system" %
%   N9:5  SYSTEM_QUICK_START %
%   B36:1/6  INITIATE_PURGE %
%   N9:6  SYSTEM_PURGE %
% Rung: 38 %
SOR EQU N10:0 N9:5 XIC S:1/15 MOV N9:1 N10:0 EOR
%   N10:0  SYSTEM_STATE  "STATE The current state of the system" %
%   N9:5  SYSTEM_QUICK_START %
%   S:1/15  FIRST_PASS  "First Pass" %
%   N9:1  SYSTEM_STANDBY  "STATE System Process" %
% Rung: 39 %
SOR EQU N10:0 N9:5 EQU N21:0 N9:118 MOV N9:2 N10:0 EOR
%   N10:0  SYSTEM_STATE  "STATE The current state of the system" %
%   N9:5  SYSTEM_QUICK_START %
%   N21:0  START_STATE %
%   N9:118  START_DONE %
%   N9:2  SYSTEM_PROCESS  "STATE System Process" %

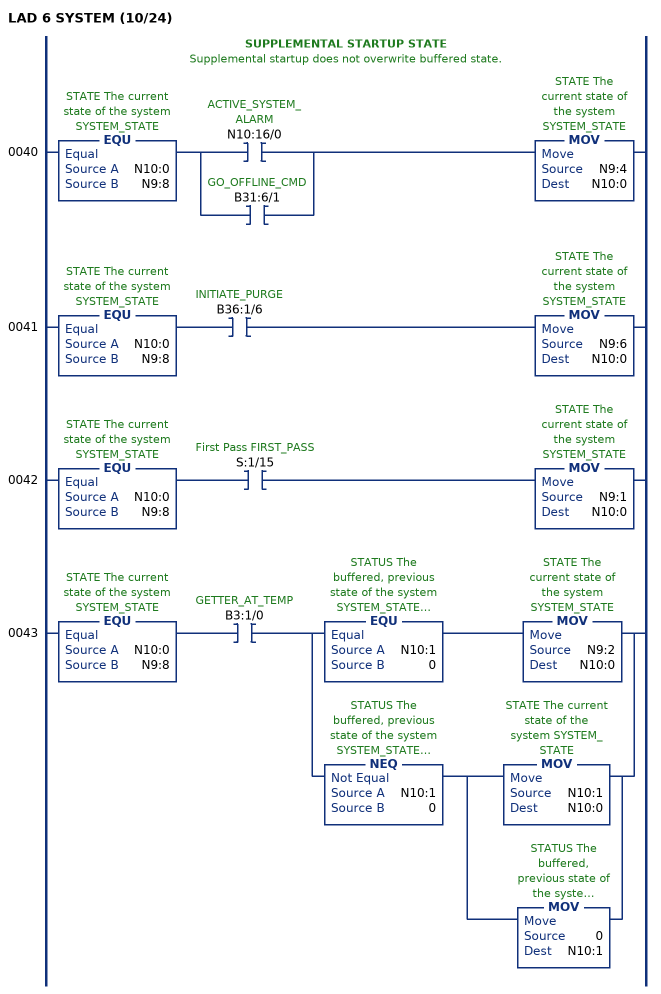
% Rung: 40 %
% TITLE: SUPPLEMENTAL STARTUP STATE %
% Supplemental startup does not overwrite buffered state. %
SOR EQU N10:0 N9:8 BST XIC N10:16/0 NXB XIC B31:6/1 BND MOV N9:4 N10:0 EOR
%   N10:0  SYSTEM_STATE  "STATE The current state of the system" %
%   N9:8  SYSTEM_SUPPLEMENTAL %
%   N10:16/0  ACTIVE_SYSTEM_ALARM %
%   B31:6/1  GO_OFFLINE_CMD %
%   N9:4  SYSTEM_ALARM  "STATE System Alarm" %
% Rung: 41 %
SOR EQU N10:0 N9:8 XIC B36:1/6 MOV N9:6 N10:0 EOR
%   N10:0  SYSTEM_STATE  "STATE The current state of the system" %
%   N9:8  SYSTEM_SUPPLEMENTAL %
%   B36:1/6  INITIATE_PURGE %
%   N9:6  SYSTEM_PURGE %
% Rung: 42 %
SOR EQU N10:0 N9:8 XIC S:1/15 MOV N9:1 N10:0 EOR
%   N10:0  SYSTEM_STATE  "STATE The current state of the system" %
%   N9:8  SYSTEM_SUPPLEMENTAL %
%   S:1/15  FIRST_PASS  "First Pass" %
%   N9:1  SYSTEM_STANDBY  "STATE System Process" %
% Rung: 43 %
SOR EQU N10:0 N9:8 XIC B3:1/0 BST EQU N10:1 0 MOV N9:2 N10:0 NXB NEQ N10:1 0 BST MOV N10:1 N10:0 NXB MOV 0 N10:1 BND BND EOR
%   N10:0  SYSTEM_STATE  "STATE The current state of the system" %
%   N9:8  SYSTEM_SUPPLEMENTAL %
%   B3:1/0  GETTER_AT_TEMP %
%   N10:1  SYSTEM_STATE_BUFFER  "STATUS The buffered, previous state of the system" %
%   N9:2  SYSTEM_PROCESS  "STATE System Process" %

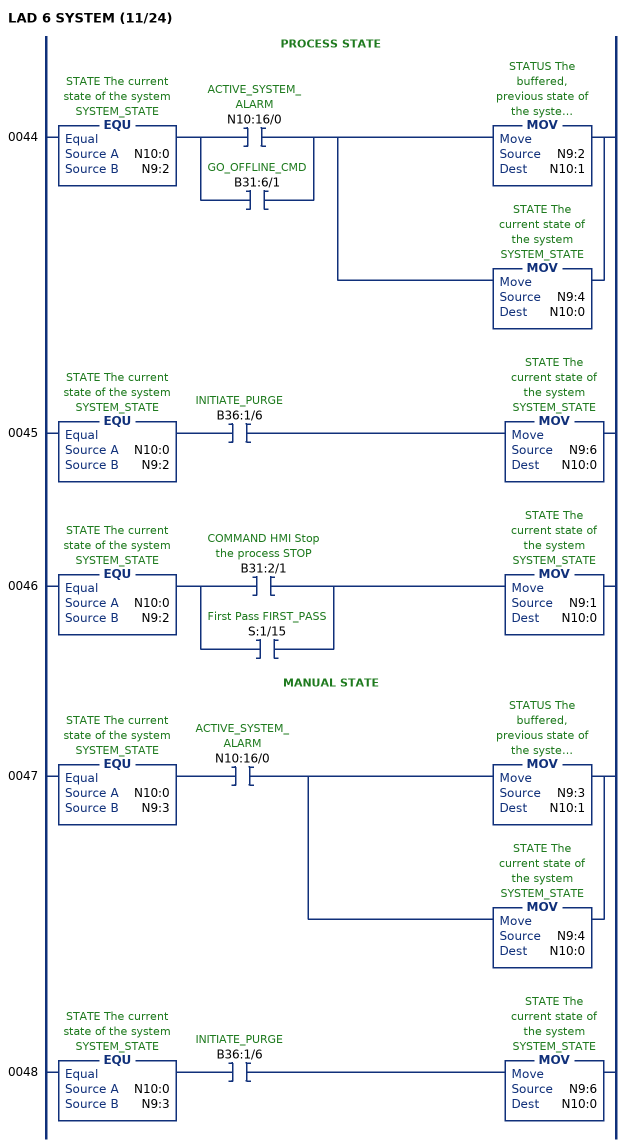
% Rung: 44 %
% TITLE: PROCESS STATE %
SOR EQU N10:0 N9:2 BST XIC N10:16/0 NXB XIC B31:6/1 BND BST MOV N9:2 N10:1 NXB MOV N9:4 N10:0 BND EOR
%   N10:0  SYSTEM_STATE  "STATE The current state of the system" %
%   N9:2  SYSTEM_PROCESS  "STATE System Process" %
%   N10:16/0  ACTIVE_SYSTEM_ALARM %
%   B31:6/1  GO_OFFLINE_CMD %
%   N10:1  SYSTEM_STATE_BUFFER  "STATUS The buffered, previous state of the system" %
%   N9:4  SYSTEM_ALARM  "STATE System Alarm" %
% Rung: 45 %
SOR EQU N10:0 N9:2 XIC B36:1/6 MOV N9:6 N10:0 EOR
%   N10:0  SYSTEM_STATE  "STATE The current state of the system" %
%   N9:2  SYSTEM_PROCESS  "STATE System Process" %
%   B36:1/6  INITIATE_PURGE %
%   N9:6  SYSTEM_PURGE %
% Rung: 46 %
SOR EQU N10:0 N9:2 BST XIC B31:2/1 NXB XIC S:1/15 BND MOV N9:1 N10:0 EOR
%   N10:0  SYSTEM_STATE  "STATE The current state of the system" %
%   N9:2  SYSTEM_PROCESS  "STATE System Process" %
%   B31:2/1  STOP  "COMMAND HMI Stop the process" %
%   S:1/15  FIRST_PASS  "First Pass" %
%   N9:1  SYSTEM_STANDBY  "STATE System Process" %
% Rung: 47 %
% TITLE: MANUAL STATE %
SOR EQU N10:0 N9:3 XIC N10:16/0 BST MOV N9:3 N10:1 NXB MOV N9:4 N10:0 BND EOR
%   N10:0  SYSTEM_STATE  "STATE The current state of the system" %
%   N9:3  SYSTEM_MANUAL  "STATE System Manual" %
%   N10:16/0  ACTIVE_SYSTEM_ALARM %
%   N10:1  SYSTEM_STATE_BUFFER  "STATUS The buffered, previous state of the system" %
%   N9:4  SYSTEM_ALARM  "STATE System Alarm" %
% Rung: 48 %
SOR EQU N10:0 N9:3 XIC B36:1/6 MOV N9:6 N10:0 EOR
%   N10:0  SYSTEM_STATE  "STATE The current state of the system" %
%   N9:3  SYSTEM_MANUAL  "STATE System Manual" %
%   B36:1/6  INITIATE_PURGE %
%   N9:6  SYSTEM_PURGE %

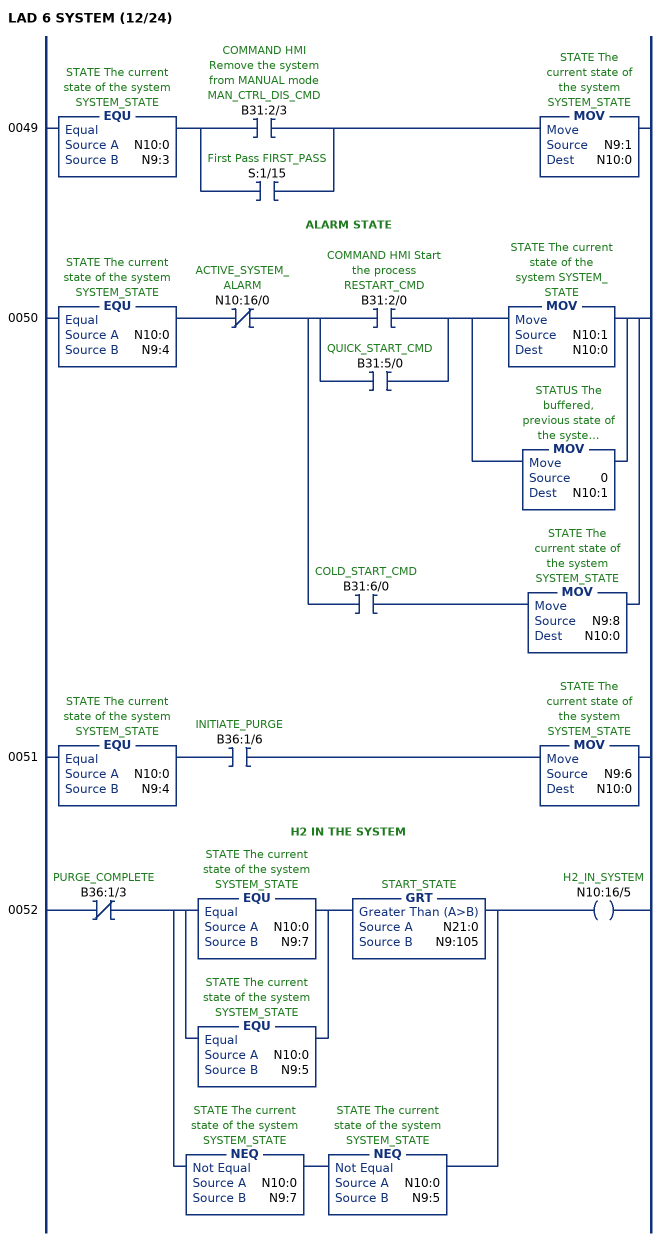
% Rung: 49 %
SOR EQU N10:0 N9:3 BST XIC B31:2/3 NXB XIC S:1/15 BND MOV N9:1 N10:0 EOR
%   N10:0  SYSTEM_STATE  "STATE The current state of the system" %
%   N9:3  SYSTEM_MANUAL  "STATE System Manual" %
%   B31:2/3  MAN_CTRL_DIS_CMD  "COMMAND HMI Remove the system from MANUAL mode" %
%   S:1/15  FIRST_PASS  "First Pass" %
%   N9:1  SYSTEM_STANDBY  "STATE System Process" %
% Rung: 50 %
% TITLE: ALARM STATE %
SOR EQU N10:0 N9:4 XIO N10:16/0 BST BST XIC B31:2/0 NXB XIC B31:5/0 BND BST MOV N10:1 N10:0 NXB MOV 0 N10:1 BND NXB XIC B31:6/0 MOV N9:8 N10:0 BND EOR
%   N10:0  SYSTEM_STATE  "STATE The current state of the system" %
%   N9:4  SYSTEM_ALARM  "STATE System Alarm" %
%   N10:16/0  ACTIVE_SYSTEM_ALARM %
%   B31:2/0  RESTART_CMD  "COMMAND HMI Start the process" %
%   B31:5/0  QUICK_START_CMD %
%   N10:1  SYSTEM_STATE_BUFFER  "STATUS The buffered, previous state of the system" %
%   B31:6/0  COLD_START_CMD %
%   N9:8  SYSTEM_SUPPLEMENTAL %
% Rung: 51 %
SOR EQU N10:0 N9:4 XIC B36:1/6 MOV N9:6 N10:0 EOR
%   N10:0  SYSTEM_STATE  "STATE The current state of the system" %
%   N9:4  SYSTEM_ALARM  "STATE System Alarm" %
%   B36:1/6  INITIATE_PURGE %
%   N9:6  SYSTEM_PURGE %
% Rung: 52 %
% TITLE: H2 IN THE SYSTEM %
SOR XIO B36:1/3 BST BST EQU N10:0 N9:7 NXB EQU N10:0 N9:5 BND GRT N21:0 N9:105 NXB NEQ N10:0 N9:7 NEQ N10:0 N9:5 BND OTE N10:16/5 EOR
%   B36:1/3  PURGE_COMPLETE %
%   N10:0  SYSTEM_STATE  "STATE The current state of the system" %
%   N9:7  SYSTEM_COLD_START %
%   N9:5  SYSTEM_QUICK_START %
%   N21:0  START_STATE %
%   N9:105  START_VENT_ALL %
%   N10:16/5  H2_IN_SYSTEM %

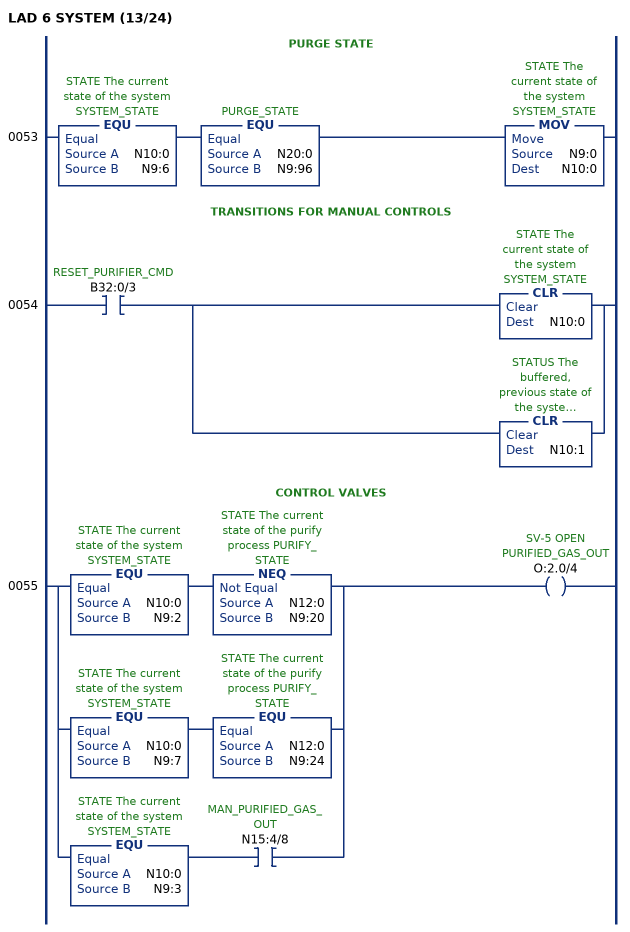
% Rung: 53 %
% TITLE: PURGE STATE %
SOR EQU N10:0 N9:6 EQU N20:0 N9:96 MOV N9:0 N10:0 EOR
%   N10:0  SYSTEM_STATE  "STATE The current state of the system" %
%   N9:6  SYSTEM_PURGE %
%   N20:0  PURGE_STATE %
%   N9:96  PURGE_DONE %
%   N9:0  SYSTEM_OFFLINE %
% Rung: 54 %
% TITLE: TRANSITIONS FOR MANUAL CONTROLS %
SOR XIC B32:0/3 BST CLR N10:0 NXB CLR N10:1 BND EOR
%   B32:0/3  RESET_PURIFIER_CMD %
%   N10:0  SYSTEM_STATE  "STATE The current state of the system" %
%   N10:1  SYSTEM_STATE_BUFFER  "STATUS The buffered, previous state of the system" %
% Rung: 55 %
% TITLE: CONTROL VALVES %
SOR BST EQU N10:0 N9:2 NEQ N12:0 N9:20 NXB EQU N10:0 N9:7 EQU N12:0 N9:24 NXB EQU N10:0 N9:3 XIC N15:4/8 BND OTE O:2.0/4 EOR
%   N10:0  SYSTEM_STATE  "STATE The current state of the system" %
%   N9:2  SYSTEM_PROCESS  "STATE System Process" %
%   N12:0  PURIFY_STATE  "STATE The current state of the purify process" %
%   N9:20  PURIFY_STANDBY  "STATE Purify Standby" %
%   N9:7  SYSTEM_COLD_START %
%   N9:24  PURIFY_OVERLAP  "STATE Puriify Overlap" %
%   N9:3  SYSTEM_MANUAL  "STATE System Manual" %
%   N15:4/8  MAN_PURIFIED_GAS_OUT %
%   O:2.0/4  PURIFIED_GAS_OUT  "SV-5 OPEN" %

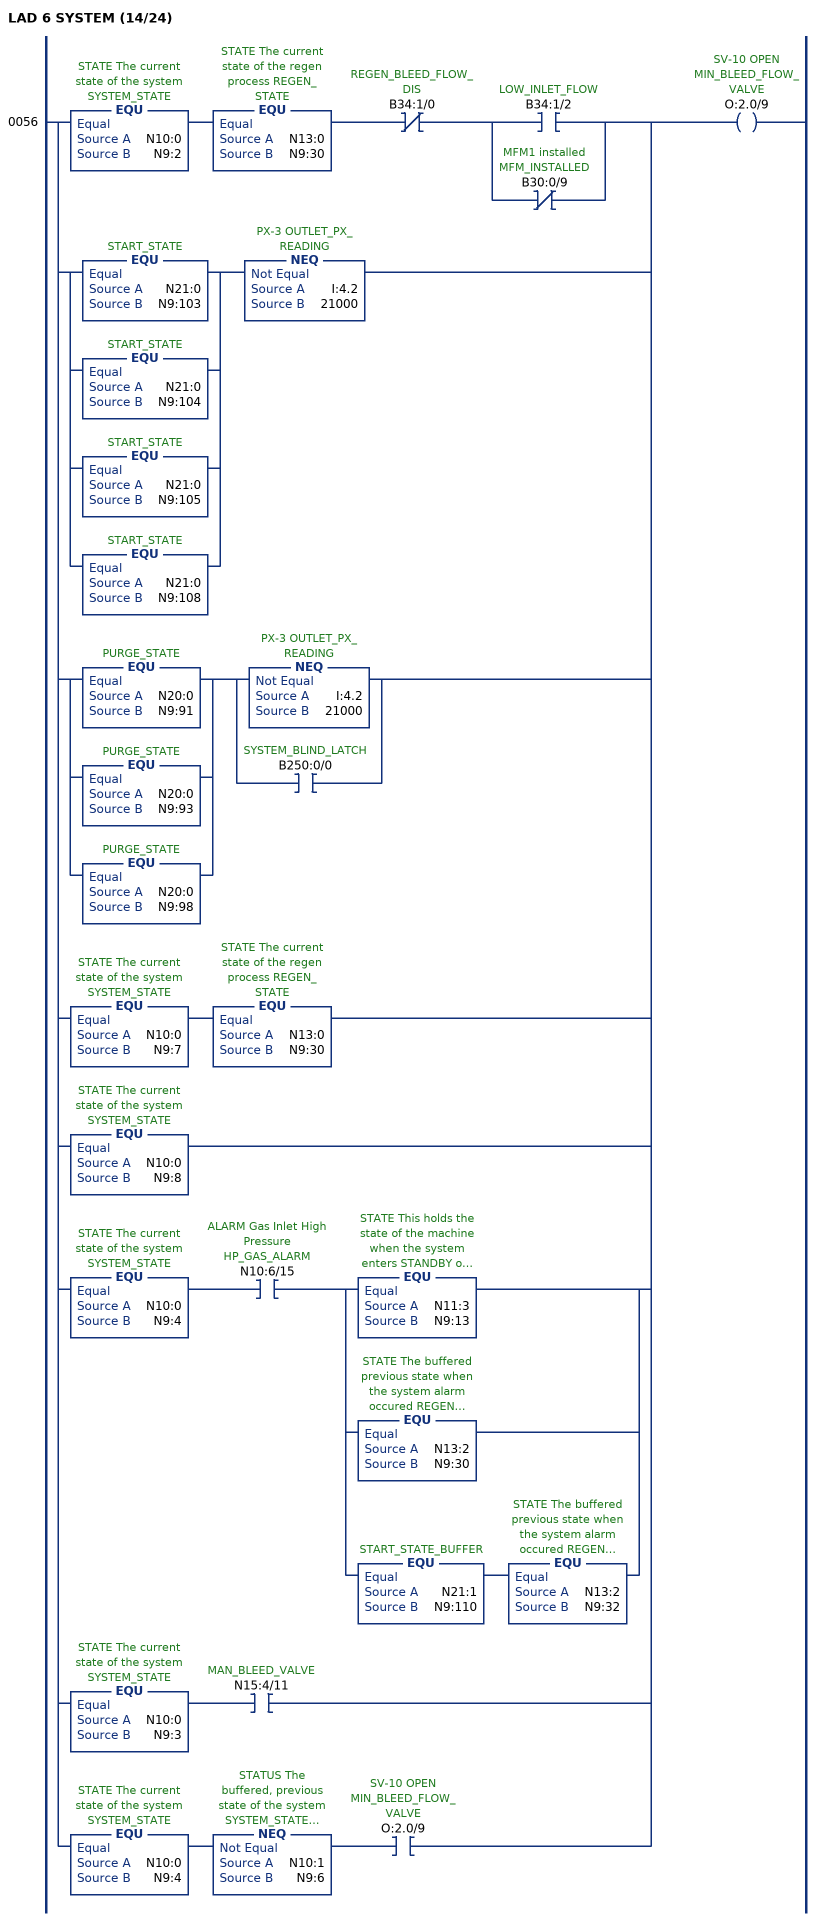
% Rung: 56 %
SOR BST EQU N10:0 N9:2 EQU N13:0 N9:30 XIO B34:1/0 BST XIC B34:1/2 NXB XIO B30:0/9 BND NXB BST EQU N21:0 N9:103 NXB EQU N21:0 N9:104 NXB EQU N21:0 N9:105 NXB EQU N21:0 N9:108 BND NEQ I:4.2 21000 NXB BST EQU N20:0 N9:91 NXB EQU N20:0 N9:93 NXB EQU N20:0 N9:98 BND BST NEQ I:4.2 21000 NXB XIC B250:0/0 BND NXB EQU N10:0 N9:7 EQU N13:0 N9:30 NXB EQU N10:0 N9:8 NXB EQU N10:0 N9:4 XIC N10:6/15 BST EQU N11:3 N9:13 NXB EQU N13:2 N9:30 NXB EQU N21:1 N9:110 EQU N13:2 N9:32 BND NXB EQU N10:0 N9:3 XIC N15:4/11 NXB EQU N10:0 N9:4 NEQ N10:1 N9:6 XIC O:2.0/9 BND OTE O:2.0/9 EOR
%   N10:0  SYSTEM_STATE  "STATE The current state of the system" %
%   N9:2  SYSTEM_PROCESS  "STATE System Process" %
%   N13:0  REGEN_STATE  "STATE The current state of the regen process" %
%   N9:30  REGEN_STANDBY  "STATE Regen Standby" %
%   B34:1/0  REGEN_BLEED_FLOW_DIS %
%   B34:1/2  LOW_INLET_FLOW %
%   B30:0/9  MFM_INSTALLED  "MFM1 installed" %
%   N21:0  START_STATE %
%   N9:103  START_VENT_GET_1 %
%   N9:104  START_HEAT %
%   N9:105  START_VENT_ALL %
%   N9:108  START_VENT_GET_2 %
%   I:4.2  OUTLET_PX_READING  "PX-3" %
%   N20:0  PURGE_STATE %
%   N9:91  PURGE_INIT_VENT %
%   N9:93  PURGE_VENT_GETTER %
%   N9:98  PURGE_VENT_GET_2 %
%   B250:0/0  SYSTEM_BLIND_LATCH %
%   N9:7  SYSTEM_COLD_START %
%   N9:8  SYSTEM_SUPPLEMENTAL %
%   N9:4  SYSTEM_ALARM  "STATE System Alarm" %
%   N10:6/15  HP_GAS_ALARM  "ALARM Gas Inlet High Pressure" %
%   N11:3  PROC_STATE_BUFFER  "STATE This holds the state of the machine when the system enters STANDBY or ALARM" %
%   N9:13  PROC_OVERLAP  "STATE Process Purify Overlap" %
%   N13:2  REGEN_SYSTEM_BUFFER  "STATE The buffered previous state when the system alarm occured" %
%   N21:1  START_STATE_BUFFER %
%   N9:110  START_REG_VENT %
%   N9:32  REGEN_VENT  "STATE Regen Vent" %
%   N9:3  SYSTEM_MANUAL  "STATE System Manual" %
%   N15:4/11  MAN_BLEED_VALVE %
%   N10:1  SYSTEM_STATE_BUFFER  "STATUS The buffered, previous state of the system" %
%   N9:6  SYSTEM_PURGE %
%   O:2.0/9  MIN_BLEED_FLOW_VALVE  "SV-10 OPEN" %

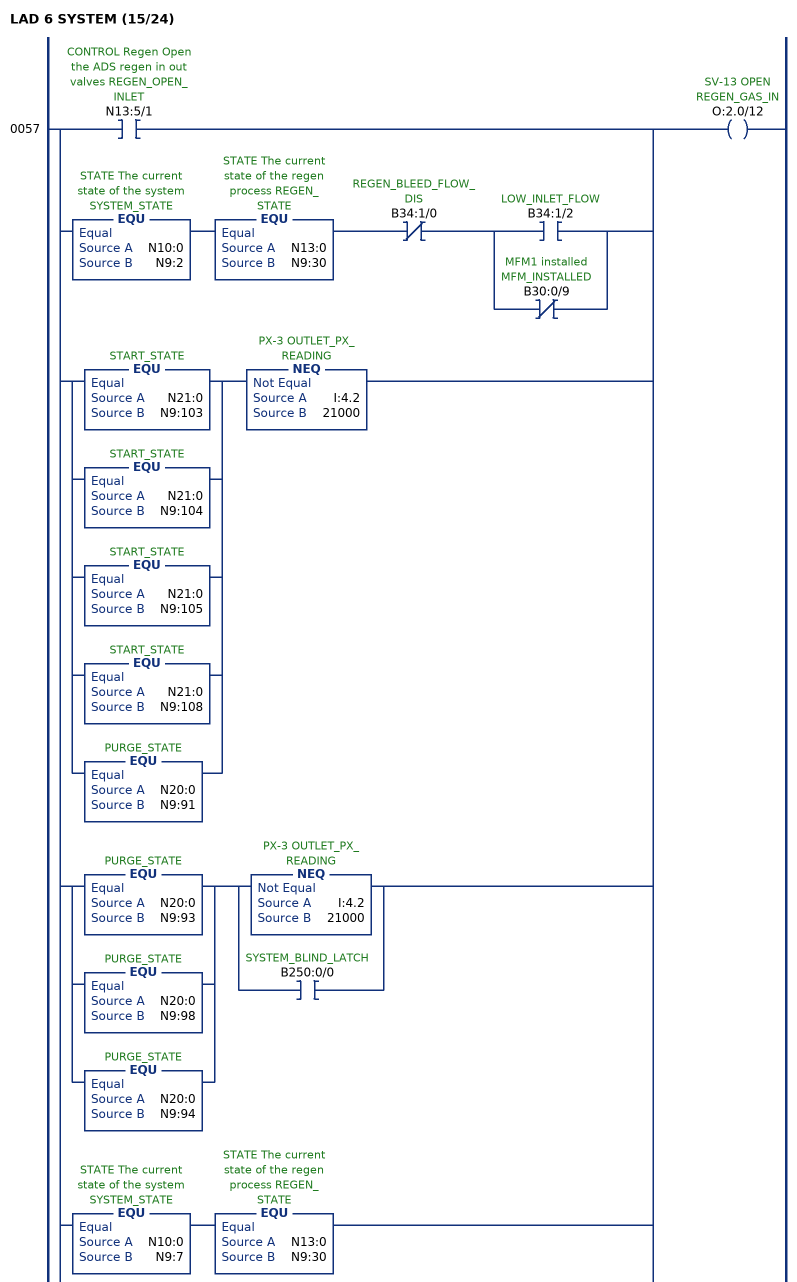

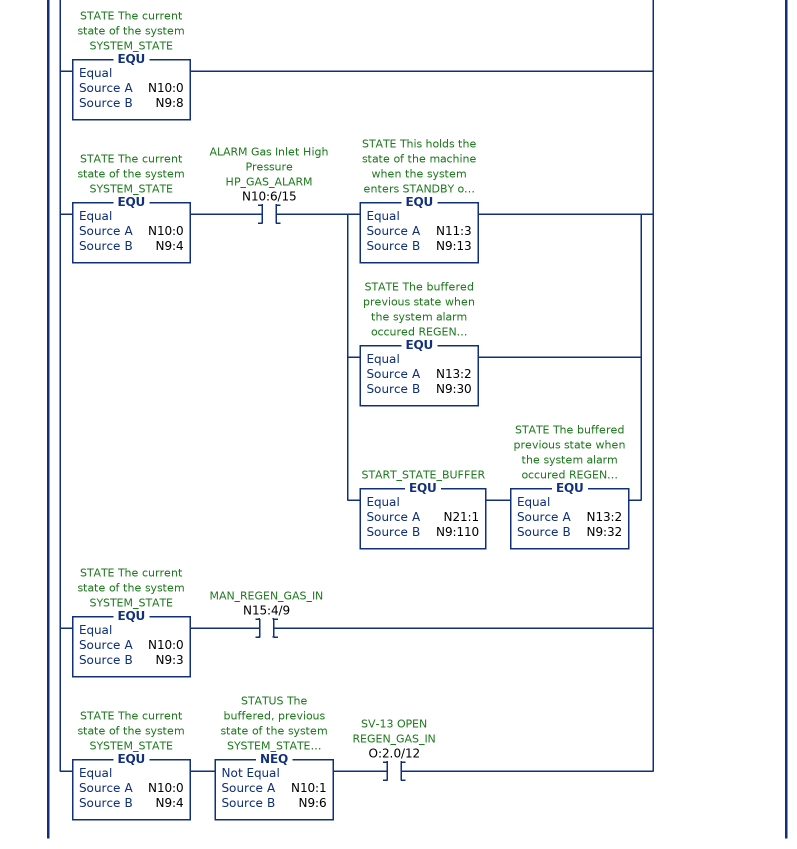
% Rung: 57 %
SOR BST XIC N13:5/1 NXB EQU N10:0 N9:2 EQU N13:0 N9:30 XIO B34:1/0 BST XIC B34:1/2 NXB XIO B30:0/9 BND NXB BST EQU N21:0 N9:103 NXB EQU N21:0 N9:104 NXB EQU N21:0 N9:105 NXB EQU N21:0 N9:108 NXB EQU N20:0 N9:91 BND NEQ I:4.2 21000 NXB BST EQU N20:0 N9:93 NXB EQU N20:0 N9:98 NXB EQU N20:0 N9:94 BND BST NEQ I:4.2 21000 NXB XIC B250:0/0 BND NXB EQU N10:0 N9:7 EQU N13:0 N9:30 NXB EQU N10:0 N9:8 NXB EQU N10:0 N9:4 XIC N10:6/15 BST EQU N11:3 N9:13 NXB EQU N13:2 N9:30 NXB EQU N21:1 N9:110 EQU N13:2 N9:32 BND NXB EQU N10:0 N9:3 XIC N15:4/9 NXB EQU N10:0 N9:4 NEQ N10:1 N9:6 XIC O:2.0/12 BND OTE O:2.0/12 EOR
%   N13:5/1  REGEN_OPEN_INLET  "CONTROL Regen Open the ADS regen in out valves" %
%   N10:0  SYSTEM_STATE  "STATE The current state of the system" %
%   N9:2  SYSTEM_PROCESS  "STATE System Process" %
%   N13:0  REGEN_STATE  "STATE The current state of the regen process" %
%   N9:30  REGEN_STANDBY  "STATE Regen Standby" %
%   B34:1/0  REGEN_BLEED_FLOW_DIS %
%   B34:1/2  LOW_INLET_FLOW %
%   B30:0/9  MFM_INSTALLED  "MFM1 installed" %
%   N21:0  START_STATE %
%   N9:103  START_VENT_GET_1 %
%   N9:104  START_HEAT %
%   N9:105  START_VENT_ALL %
%   N9:108  START_VENT_GET_2 %
%   N20:0  PURGE_STATE %
%   N9:91  PURGE_INIT_VENT %
%   I:4.2  OUTLET_PX_READING  "PX-3" %
%   N9:93  PURGE_VENT_GETTER %
%   N9:98  PURGE_VENT_GET_2 %
%   N9:94  PURGE_BACKFILL %
%   B250:0/0  SYSTEM_BLIND_LATCH %
%   N9:7  SYSTEM_COLD_START %
%   N9:8  SYSTEM_SUPPLEMENTAL %
%   N9:4  SYSTEM_ALARM  "STATE System Alarm" %
%   N10:6/15  HP_GAS_ALARM  "ALARM Gas Inlet High Pressure" %
%   N11:3  PROC_STATE_BUFFER  "STATE This holds the state of the machine when the system enters STANDBY or ALARM" %
%   N9:13  PROC_OVERLAP  "STATE Process Purify Overlap" %
%   N13:2  REGEN_SYSTEM_BUFFER  "STATE The buffered previous state when the system alarm occured" %
%   N21:1  START_STATE_BUFFER %
%   N9:110  START_REG_VENT %
%   N9:32  REGEN_VENT  "STATE Regen Vent" %
%   N9:3  SYSTEM_MANUAL  "STATE System Manual" %
%   N15:4/9  MAN_REGEN_GAS_IN %
%   N10:1  SYSTEM_STATE_BUFFER  "STATUS The buffered, previous state of the system" %
%   N9:6  SYSTEM_PURGE %
%   O:2.0/12  REGEN_GAS_IN  "SV-13 OPEN" %

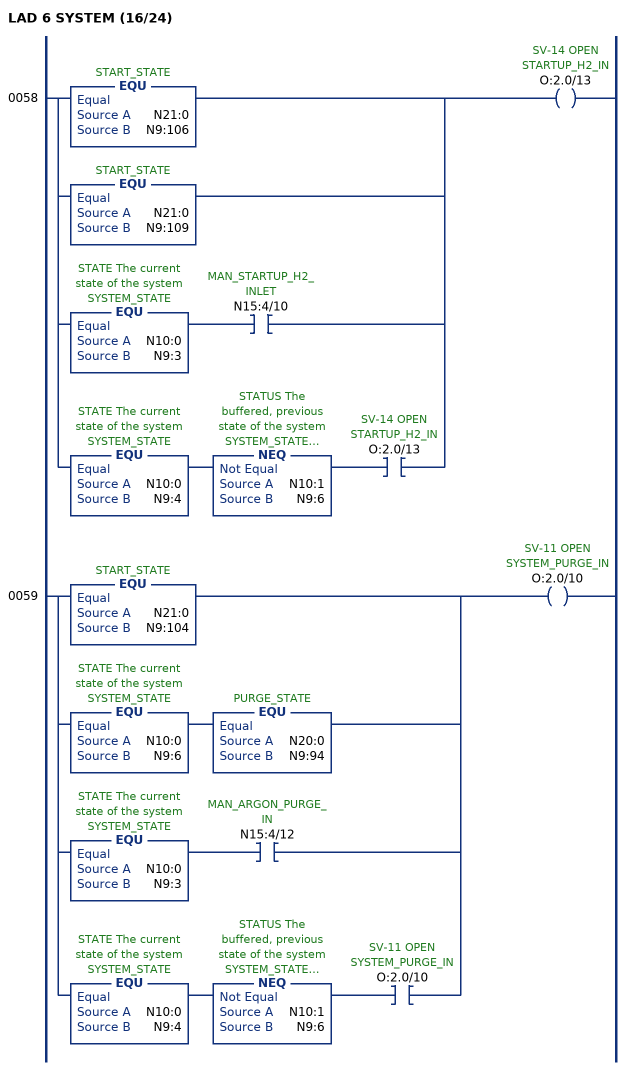
% Rung: 58 %
SOR BST BST EQU N21:0 N9:106 NXB EQU N21:0 N9:109 BND NXB EQU N10:0 N9:3 XIC N15:4/10 NXB EQU N10:0 N9:4 NEQ N10:1 N9:6 XIC O:2.0/13 BND OTE O:2.0/13 EOR
%   N21:0  START_STATE %
%   N9:106  START_BACKFILL_1 %
%   N9:109  START_BACKFILL_2 %
%   N10:0  SYSTEM_STATE  "STATE The current state of the system" %
%   N9:3  SYSTEM_MANUAL  "STATE System Manual" %
%   N15:4/10  MAN_STARTUP_H2_INLET %
%   N9:4  SYSTEM_ALARM  "STATE System Alarm" %
%   N10:1  SYSTEM_STATE_BUFFER  "STATUS The buffered, previous state of the system" %
%   N9:6  SYSTEM_PURGE %
%   O:2.0/13  STARTUP_H2_IN  "SV-14 OPEN" %
% Rung: 59 %
SOR BST EQU N21:0 N9:104 NXB EQU N10:0 N9:6 EQU N20:0 N9:94 NXB EQU N10:0 N9:3 XIC N15:4/12 NXB EQU N10:0 N9:4 NEQ N10:1 N9:6 XIC O:2.0/10 BND OTE O:2.0/10 EOR
%   N21:0  START_STATE %
%   N9:104  START_HEAT %
%   N10:0  SYSTEM_STATE  "STATE The current state of the system" %
%   N9:6  SYSTEM_PURGE %
%   N20:0  PURGE_STATE %
%   N9:94  PURGE_BACKFILL %
%   N9:3  SYSTEM_MANUAL  "STATE System Manual" %
%   N15:4/12  MAN_ARGON_PURGE_IN %
%   N9:4  SYSTEM_ALARM  "STATE System Alarm" %
%   N10:1  SYSTEM_STATE_BUFFER  "STATUS The buffered, previous state of the system" %
%   O:2.0/10  SYSTEM_PURGE_IN  "SV-11 OPEN" %

